LIN {X 0,Y 573.258,Z 350.075,A -85,B 0,C 180,E1 -2304.01,E2 -2304.01} C_VEL
LIN {X 0,Y 573.278,Z 350.069,A -85,B 0,C 180,E1 -2306.518,E2 -2306.518} C_VEL
LIN {X 0,Y 573.237,Z 350.079,A -85,B 0,C 180,E1 -2309.114,E2 -2309.114} C_VEL
LIN {X 0,Y 573.258,Z 350.074,A -85,B 0,C 180,E1 -2311.968,E2 -2311.968} C_VEL
LIN {X 0,Y 573.248,Z 350.071,A -85,B 0,C 180,E1 -2314.59,E2 -2314.59} C_VEL
LIN {X 0,Y 573.251,Z 350.077,A -85,B 0,C 180,E1 -2317.663,E2 -2317.663} C_VEL
LIN {X 0,Y 573.27,Z 350.072,A -85,B 0,C 180,E1 -2320.727,E2 -2320.727} C_VEL
LIN {X 0,Y 573.253,Z 350.076,A -85,B 0,C 180,E1 -2323.622,E2 -2323.622} C_VEL
LIN {X 0,Y 573.232,Z 350.077,A -85,B 0,C 180,E1 -2326.53,E2 -2326.53} C_VEL
LIN {X 0,Y 573.269,Z 350.075,A -85,B 0,C 180,E1 -2329.404,E2 -2329.404} C_VEL
LIN {X 0,Y 573.282,Z 350.069,A -85,B 0,C 180,E1 -2332.25,E2 -2332.25} C_VEL
LIN {X 0,Y 573.307,Z 350.074,A -85,B 0,C 180,E1 -2335.077,E2 -2335.077} C_VEL
LIN {X 0,Y 573.301,Z 350.066,A -85,B 0,C 180,E1 -2337.893,E2 -2337.893} C_VEL
LIN {X 0,Y 573.334,Z 350.07,A -85,B 0,C 180,E1 -2340.703,E2 -2340.703} C_VEL
LIN {X 0,Y 573.237,Z 350.074,A -85,B 0,C 180,E1 -2343.515,E2 -2343.515} C_VEL
LIN {X 0,Y 573.286,Z 350.069,A -85,B 0,C 180,E1 -2345.628,E2 -2345.628} C_VEL
LIN {X 0,Y 573.3,Z 350.072,A -85,B 0,C 180,E1 -2348.459,E2 -2348.459} C_VEL
LIN {X 0,Y 573.29,Z 350.069,A -85,B 0,C 180,E1 -2351.312,E2 -2351.312} C_VEL
LIN {X 0,Y 573.272,Z 350.077,A -85,B 0,C 180,E1 -2354.425,E2 -2354.425} C_VEL
LIN {X 0,Y 573.252,Z 350.074,A -85,B 0,C 180,E1 -2357.112,E2 -2357.112} C_VEL
LIN {X 0,Y 573.249,Z 350.077,A -85,B 0,C 180,E1 -2360.077,E2 -2360.077} C_VEL
LIN {X 0,Y 573.232,Z 350.084,A -85,B 0,C 180,E1 -2362.338,E2 -2362.338} C_VEL
LIN {X 0,Y 573.244,Z 350.076,A -85,B 0,C 180,E1 -2364.406,E2 -2364.406} C_VEL
LIN {X 0,Y 572.619,Z 350.155,A -85,B 0,C 180,E1 -2364.993,E2 -2364.993} C_VEL
LIN {X 0,Y 569.78,Z 350.507,A -85,B 0,C 180,E1 -2365.944,E2 -2365.944} C_VEL
LIN {X 0,Y 567.351,Z 350.81,A -85,B 0,C 180,E1 -2366.71,E2 -2366.71} C_VEL
LIN {X 0,Y 566.299,Z 350.937,A -85,B 0,C 180,E1 -2367.301,E2 -2367.301} C_VEL
LIN {X 0,Y 566.21,Z 350.948,A -85,B 0,C 180,E1 -2367.502,E2 -2367.502} C_VEL
LIN {X 0,Y 566.182,Z 350.957,A -85,B 0,C 180,E1 -2370.593,E2 -2370.593} C_VEL
LIN {X 0,Y 566.224,Z 350.948,A -85,B 0,C 180,E1 -2373.102,E2 -2373.102} C_VEL
LIN {X 0,Y 566.207,Z 350.954,A -85,B 0,C 180,E1 -2375.689,E2 -2375.689} C_VEL
LIN {X 0,Y 566.213,Z 350.953,A -85,B 0,C 180,E1 -2378.56,E2 -2378.56} C_VEL
LIN {X 0,Y 566.21,Z 350.951,A -85,B 0,C 180,E1 -2381.137,E2 -2381.137} C_VEL
LIN {X 0,Y 566.198,Z 350.962,A -85,B 0,C 180,E1 -2384.036,E2 -2384.036} C_VEL
LIN {X 0,Y 566.203,Z 350.952,A -85,B 0,C 180,E1 -2387.083,E2 -2387.083} C_VEL
LIN {X 0,Y 566.227,Z 350.958,A -85,B 0,C 180,E1 -2389.804,E2 -2389.804} C_VEL
LIN {X 0,Y 566.2,Z 350.952,A -85,B 0,C 180,E1 -2392.6,E2 -2392.6} C_VEL
LIN {X 0,Y 566.223,Z 350.951,A -85,B 0,C 180,E1 -2395.184,E2 -2395.184} C_VEL
LIN {X 0,Y 566.234,Z 350.956,A -85,B 0,C 180,E1 -2397.744,E2 -2397.744} C_VEL
LIN {X 0,Y 566.231,Z 350.95,A -85,B 0,C 180,E1 -2400.324,E2 -2400.324} C_VEL
LIN {X 0,Y 566.246,Z 351.051,A -85,B 0,C 180,E1 -2402.588,E2 -2402.588} C_VEL
LIN {X 0,Y 566.363,Z 357.712,A -85,B 0,C 180,E1 -2403.864,E2 -2403.864} C_VEL
LIN {X 0,Y 566.226,Z 372.791,A -85,B 0,C 180,E1 -2406.707,E2 -2406.707} C_VEL
LIN {X 0,Y 566.214,Z 374.601,A -85,B 0,C 180,E1 -2407.046,E2 -2407.046} C_VEL
LIN {X 0,Y 567.183,Z 380.548,A -85,B 0,C 180,E1 -2407.157,E2 -2407.157} C_VEL
LIN {X 0,Y 566.926,Z 481.627,A -85,B 0,C 180,E1 -2408.461,E2 -2408.461} C_VEL
LIN {X 0,Y 566.83,Z 495.188,A -85,B 0,C 180,E1 -2408.793,E2 -2408.793} C_VEL
LIN {X 0,Y 566.692,Z 507.886,A -85,B 0,C 180,E1 -2409.254,E2 -2409.254} C_VEL
LIN {X 0,Y 566.578,Z 520.156,A -85,B 0,C 180,E1 -2409.866,E2 -2409.866} C_VEL
LIN {X 0,Y 566.42,Z 531.079,A -85,B 0,C 180,E1 -2410.561,E2 -2410.561} C_VEL
LIN {X 0,Y 566.291,Z 541.23,A -85,B 0,C 180,E1 -2411.363,E2 -2411.363} C_VEL
LIN {X 0,Y 566.183,Z 550.756,A -85,B 0,C 180,E1 -2412.295,E2 -2412.295} C_VEL
LIN {X 0,Y 566.05,Z 559.938,A -85,B 0,C 180,E1 -2413.408,E2 -2413.408} C_VEL
LIN {X 0,Y 566.009,Z 567.237,A -85,B 0,C 180,E1 -2414.517,E2 -2414.517} C_VEL
LIN {X 0,Y 565.941,Z 572.998,A -85,B 0,C 180,E1 -2415.62,E2 -2415.62} C_VEL
LIN {X 0,Y 565.929,Z 577.491,A -85,B 0,C 180,E1 -2416.718,E2 -2416.718} C_VEL
LIN {X 0,Y 565.895,Z 580.853,A -85,B 0,C 180,E1 -2417.812,E2 -2417.812} C_VEL
LIN {X 0,Y 565.905,Z 583.1,A -85,B 0,C 180,E1 -2418.847,E2 -2418.847} C_VEL
LIN {X 0,Y 565.883,Z 584.554,A -85,B 0,C 180,E1 -2419.987,E2 -2419.987} C_VEL
LIN {X 0,Y 565.853,Z 584.921,A -85,B 0,C 180,E1 -2421.429,E2 -2421.429} C_VEL
LIN {X 0,Y 565.879,Z 584.522,A -85,B 0,C 180,E1 -2422.148,E2 -2422.148} C_VEL
LIN {X 0,Y 565.921,Z 582.681,A -85,B 0,C 180,E1 -2423.466,E2 -2423.466} C_VEL
LIN {X 0,Y 565.917,Z 579.807,A -85,B 0,C 180,E1 -2424.656,E2 -2424.656} C_VEL
LIN {X 0,Y 565.957,Z 576.164,A -85,B 0,C 180,E1 -2425.727,E2 -2425.727} C_VEL
LIN {X 0,Y 565.954,Z 571.425,A -85,B 0,C 180,E1 -2426.797,E2 -2426.797} C_VEL
LIN {X 0,Y 566.008,Z 564.341,A -85,B 0,C 180,E1 -2428.043,E2 -2428.043} C_VEL
LIN {X 0,Y 566.12,Z 556.652,A -85,B 0,C 180,E1 -2429.111,E2 -2429.111} C_VEL
LIN {X 0,Y 566.205,Z 547.068,A -85,B 0,C 180,E1 -2430.178,E2 -2430.178} C_VEL
LIN {X 0,Y 566.344,Z 537.198,A -85,B 0,C 180,E1 -2431.067,E2 -2431.067} C_VEL
LIN {X 0,Y 566.445,Z 526.095,A -85,B 0,C 180,E1 -2431.866,E2 -2431.866} C_VEL
LIN {X 0,Y 566.589,Z 515.253,A -85,B 0,C 180,E1 -2432.488,E2 -2432.488} C_VEL
LIN {X 0,Y 566.707,Z 503.304,A -85,B 0,C 180,E1 -2433.021,E2 -2433.021} C_VEL
LIN {X 0,Y 566.839,Z 490.96,A -85,B 0,C 180,E1 -2433.421,E2 -2433.421} C_VEL
LIN {X 0,Y 566.908,Z 478.202,A -85,B 0,C 180,E1 -2433.687,E2 -2433.687} C_VEL
LIN {X 0,Y 567.109,Z 380.113,A -85,B 0,C 180,E1 -2434.94,E2 -2434.94} C_VEL
LIN {X 0,Y 566.288,Z 374.554,A -85,B 0,C 180,E1 -2435.051,E2 -2435.051} C_VEL
LIN {X 0,Y 566.37,Z 357.828,A -85,B 0,C 180,E1 -2438.204,E2 -2438.204} C_VEL
LIN {X 0,Y 566.223,Z 350.954,A -85,B 0,C 180,E1 -2439.533,E2 -2439.533} C_VEL
LIN {X 0,Y 566.247,Z 350.953,A -85,B 0,C 180,E1 -2442.18,E2 -2442.18} C_VEL
LIN {X 0,Y 566.205,Z 350.951,A -85,B 0,C 180,E1 -2445.109,E2 -2445.109} C_VEL
LIN {X 0,Y 566.205,Z 350.951,A -85,B 0,C 180,E1 -2447.331,E2 -2447.331} C_VEL
LIN {X 0,Y 566.213,Z 350.959,A -85,B 0,C 180,E1 -2450.337,E2 -2450.337} C_VEL
LIN {X 0,Y 566.194,Z 350.952,A -85,B 0,C 180,E1 -2453.403,E2 -2453.403} C_VEL
LIN {X 0,Y 566.217,Z 350.952,A -85,B 0,C 180,E1 -2455.748,E2 -2455.748} C_VEL
LIN {X 0,Y 566.21,Z 350.96,A -85,B 0,C 180,E1 -2458.202,E2 -2458.202} C_VEL
LIN {X 0,Y 566.189,Z 350.956,A -85,B 0,C 180,E1 -2460.591,E2 -2460.591} C_VEL
LIN {X 0,Y 566.23,Z 350.948,A -85,B 0,C 180,E1 -2463.101,E2 -2463.101} C_VEL
LIN {X 0,Y 566.214,Z 350.955,A -85,B 0,C 180,E1 -2465.687,E2 -2465.687} C_VEL
LIN {X 0,Y 566.216,Z 350.951,A -85,B 0,C 180,E1 -2468.558,E2 -2468.558} C_VEL
LIN {X 0,Y 566.202,Z 350.952,A -85,B 0,C 180,E1 -2471.136,E2 -2471.136} C_VEL
LIN {X 0,Y 566.195,Z 350.959,A -85,B 0,C 180,E1 -2474.035,E2 -2474.035} C_VEL
LIN {X 0,Y 566.203,Z 350.952,A -85,B 0,C 180,E1 -2477.081,E2 -2477.081} C_VEL
LIN {X 0,Y 566.223,Z 350.958,A -85,B 0,C 180,E1 -2479.802,E2 -2479.802} C_VEL
LIN {X 0,Y 566.195,Z 350.953,A -85,B 0,C 180,E1 -2482.598,E2 -2482.598} C_VEL
LIN {X 0,Y 566.204,Z 350.954,A -85,B 0,C 180,E1 -2485.181,E2 -2485.181} C_VEL
LIN {X 0,Y 566.231,Z 350.956,A -85,B 0,C 180,E1 -2487.743,E2 -2487.743} C_VEL
LIN {X 0,Y 566.198,Z 350.953,A -85,B 0,C 180,E1 -2490.327,E2 -2490.327} C_VEL
LIN {X 0,Y 566.219,Z 350.95,A -85,B 0,C 180,E1 -2492.661,E2 -2492.661} C_VEL
LIN {X 0,Y 566.228,Z 350.952,A -85,B 0,C 180,E1 -2495.038,E2 -2495.038} C_VEL
LIN {X 0,Y 566.197,Z 350.96,A -85,B 0,C 180,E1 -2497.369,E2 -2497.369} C_VEL
LIN {X 0,Y 566.213,Z 350.956,A -85,B 0,C 180,E1 -2499.663,E2 -2499.663} C_VEL
LIN {X 0,Y 566.198,Z 350.954,A -85,B 0,C 180,E1 -2502.668,E2 -2502.668} C_VEL
LIN {X 0,Y 566.225,Z 350.953,A -85,B 0,C 180,E1 -2505.626,E2 -2505.626} C_VEL
LIN {X 0,Y 566.266,Z 350.946,A -85,B 0,C 180,E1 -2508.654,E2 -2508.654} C_VEL
LIN {X 0,Y 566.242,Z 350.953,A -85,B 0,C 180,E1 -2511.434,E2 -2511.434} C_VEL
LIN {X 0,Y 566.255,Z 350.946,A -85,B 0,C 180,E1 -2514.301,E2 -2514.301} C_VEL
LIN {X 0,Y 566.273,Z 350.943,A -85,B 0,C 180,E1 -2517.866,E2 -2517.866} C_VEL
LIN {X 0,Y 566.302,Z 350.945,A -85,B 0,C 180,E1 -2520.711,E2 -2520.711} C_VEL
LIN {X 0,Y 566.273,Z 350.951,A -85,B 0,C 180,E1 -2522.845,E2 -2522.845} C_VEL
LIN {X 0,Y 566.255,Z 350.946,A -85,B 0,C 180,E1 -2525.698,E2 -2525.698} C_VEL
LIN {X 0,Y 566.241,Z 350.952,A -85,B 0,C 180,E1 -2528.565,E2 -2528.565} C_VEL
LIN {X 0,Y 566.241,Z 350.948,A -85,B 0,C 180,E1 -2531.454,E2 -2531.454} C_VEL
LIN {X 0,Y 566.224,Z 350.955,A -85,B 0,C 180,E1 -2534.507,E2 -2534.507} C_VEL
LIN {X 0,Y 566.197,Z 350.954,A -85,B 0,C 180,E1 -2537.332,E2 -2537.332} C_VEL
LIN {X 0,Y 566.213,Z 350.955,A -85,B 0,C 180,E1 -2540.337,E2 -2540.337} C_VEL
LIN {X 0,Y 566.222,Z 350.95,A -85,B 0,C 180,E1 -2543.402,E2 -2543.402} C_VEL
LIN {X 0,Y 566.217,Z 350.95,A -85,B 0,C 180,E1 -2545.749,E2 -2545.749} C_VEL
LIN {X 0,Y 566.2,Z 350.957,A -85,B 0,C 180,E1 -2548.204,E2 -2548.204} C_VEL
LIN {X 0,Y 566.193,Z 350.954,A -85,B 0,C 180,E1 -2551.079,E2 -2551.079} C_VEL
LIN {X 0,Y 566.222,Z 350.95,A -85,B 0,C 180,E1 -2553.738,E2 -2553.738} C_VEL
LIN {X 0,Y 566.21,Z 350.957,A -85,B 0,C 180,E1 -2556.569,E2 -2556.569} C_VEL
LIN {X 0,Y 566.207,Z 350.952,A -85,B 0,C 180,E1 -2559.686,E2 -2559.686} C_VEL
LIN {X 0,Y 566.209,Z 350.958,A -85,B 0,C 180,E1 -2562.088,E2 -2562.088} C_VEL
LIN {X 0,Y 566.169,Z 350.956,A -85,B 0,C 180,E1 -2565.037,E2 -2565.037} C_VEL
LIN {X 0,Y 566.214,Z 350.959,A -85,B 0,C 180,E1 -2568.137,E2 -2568.137} C_VEL
LIN {X 0,Y 566.22,Z 350.95,A -85,B 0,C 180,E1 -2570.728,E2 -2570.728} C_VEL
LIN {X 0,Y 566.216,Z 350.955,A -85,B 0,C 180,E1 -2573.784,E2 -2573.784} C_VEL
LIN {X 0,Y 566.211,Z 350.955,A -85,B 0,C 180,E1 -2576.266,E2 -2576.266} C_VEL
LIN {X 0,Y 566.202,Z 350.951,A -85,B 0,C 180,E1 -2578.922,E2 -2578.922} C_VEL
LIN {X 0,Y 566.195,Z 350.953,A -85,B 0,C 180,E1 -2581.048,E2 -2581.048} C_VEL
LIN {X 0,Y 566.217,Z 350.954,A -85,B 0,C 180,E1 -2583.46,E2 -2583.46} C_VEL
LIN {X 0,Y 566.236,Z 351.046,A -85,B 0,C 180,E1 -2585.919,E2 -2585.919} C_VEL
LIN {X 0,Y 567.201,Z 357.181,A -85,B 0,C 180,E1 -2586.834,E2 -2586.834} C_VEL
LIN {X 0,Y 566.963,Z 376.072,A -85,B 0,C 180,E1 -2589.502,E2 -2589.502} C_VEL
LIN {X 0,Y 566.667,Z 397.345,A -85,B 0,C 180,E1 -2592.497,E2 -2592.497} C_VEL
LIN {X 0,Y 566.459,Z 419.948,A -85,B 0,C 180,E1 -2595.633,E2 -2595.633} C_VEL
LIN {X 0,Y 566.417,Z 422.524,A -85,B 0,C 180,E1 -2595.987,E2 -2595.987} C_VEL
LIN {X 0,Y 567.226,Z 430.323,A -85,B 0,C 180,E1 -2596.11,E2 -2596.11} C_VEL
LIN {X 0,Y 566.964,Z 530.961,A -85,B 0,C 180,E1 -2597.403,E2 -2597.403} C_VEL
LIN {X 0,Y 566.871,Z 544.228,A -85,B 0,C 180,E1 -2597.72,E2 -2597.72} C_VEL
LIN {X 0,Y 566.74,Z 556.383,A -85,B 0,C 180,E1 -2598.148,E2 -2598.148} C_VEL
LIN {X 0,Y 566.589,Z 568.449,A -85,B 0,C 180,E1 -2598.724,E2 -2598.724} C_VEL
LIN {X 0,Y 566.442,Z 580.203,A -85,B 0,C 180,E1 -2599.455,E2 -2599.455} C_VEL
LIN {X 0,Y 566.321,Z 590.605,A -85,B 0,C 180,E1 -2600.266,E2 -2600.266} C_VEL
LIN {X 0,Y 566.207,Z 599.115,A -85,B 0,C 180,E1 -2601.074,E2 -2601.074} C_VEL
LIN {X 0,Y 566.112,Z 606.962,A -85,B 0,C 180,E1 -2601.972,E2 -2601.972} C_VEL
LIN {X 0,Y 566.003,Z 614.623,A -85,B 0,C 180,E1 -2603.047,E2 -2603.047} C_VEL
LIN {X 0,Y 566.004,Z 621.68,A -85,B 0,C 180,E1 -2604.299,E2 -2604.299} C_VEL
LIN {X 0,Y 565.933,Z 626.373,A -85,B 0,C 180,E1 -2605.37,E2 -2605.37} C_VEL
LIN {X 0,Y 565.927,Z 629.958,A -85,B 0,C 180,E1 -2606.44,E2 -2606.44} C_VEL
LIN {X 0,Y 565.878,Z 631.808,A -85,B 0,C 180,E1 -2607.153,E2 -2607.153} C_VEL
LIN {X 0,Y 565.846,Z 634.185,A -85,B 0,C 180,E1 -2608.577,E2 -2608.577} C_VEL
LIN {X 0,Y 565.839,Z 635,A -85,B 0,C 180,E1 -2610,E2 -2610} C_VEL
LIN {X 0,Y 565.846,Z 634.186,A -85,B 0,C 180,E1 -2611.423,E2 -2611.423} C_VEL
LIN {X 0,Y 565.878,Z 631.81,A -85,B 0,C 180,E1 -2612.847,E2 -2612.847} C_VEL
LIN {X 0,Y 565.926,Z 628.896,A -85,B 0,C 180,E1 -2613.916,E2 -2613.916} C_VEL
LIN {X 0,Y 565.878,Z 624.949,A -85,B 0,C 180,E1 -2614.987,E2 -2614.987} C_VEL
LIN {X 0,Y 566.002,Z 619.868,A -85,B 0,C 180,E1 -2616.058,E2 -2616.058} C_VEL
LIN {X 0,Y 566.04,Z 613.469,A -85,B 0,C 180,E1 -2617.132,E2 -2617.132} C_VEL
LIN {X 0,Y 566.133,Z 605.479,A -85,B 0,C 180,E1 -2618.207,E2 -2618.207} C_VEL
LIN {X 0,Y 566.228,Z 597.337,A -85,B 0,C 180,E1 -2619.105,E2 -2619.105} C_VEL
LIN {X 0,Y 566.343,Z 587.403,A -85,B 0,C 180,E1 -2620.005,E2 -2620.005} C_VEL
LIN {X 0,Y 566.529,Z 576.294,A -85,B 0,C 180,E1 -2620.807,E2 -2620.807} C_VEL
LIN {X 0,Y 566.612,Z 565.181,A -85,B 0,C 180,E1 -2621.446,E2 -2621.446} C_VEL
LIN {X 0,Y 566.736,Z 552.989,A -85,B 0,C 180,E1 -2621.988,E2 -2621.988} C_VEL
LIN {X 0,Y 566.91,Z 540.187,A -85,B 0,C 180,E1 -2622.393,E2 -2622.393} C_VEL
LIN {X 0,Y 566.997,Z 528.125,A -85,B 0,C 180,E1 -2622.641,E2 -2622.641} C_VEL
LIN {X 0,Y 567.065,Z 426.951,A -85,B 0,C 180,E1 -2623.937,E2 -2623.937} C_VEL
LIN {X 0,Y 566.435,Z 422.441,A -85,B 0,C 180,E1 -2624.024,E2 -2624.024} C_VEL
LIN {X 0,Y 566.648,Z 399.148,A -85,B 0,C 180,E1 -2627.251,E2 -2627.251} C_VEL
LIN {X 0,Y 566.926,Z 378.732,A -85,B 0,C 180,E1 -2630.121,E2 -2630.121} C_VEL
LIN {X 0,Y 567.199,Z 357.121,A -85,B 0,C 180,E1 -2633.166,E2 -2633.166} C_VEL
LIN {X 0,Y 566.236,Z 350.957,A -85,B 0,C 180,E1 -2634.105,E2 -2634.105} C_VEL
LIN {X 0,Y 566.209,Z 350.954,A -85,B 0,C 180,E1 -2636.659,E2 -2636.659} C_VEL
LIN {X 0,Y 566.195,Z 350.953,A -85,B 0,C 180,E1 -2638.952,E2 -2638.952} C_VEL
LIN {X 0,Y 566.202,Z 350.952,A -85,B 0,C 180,E1 -2641.42,E2 -2641.42} C_VEL
LIN {X 0,Y 566.211,Z 350.959,A -85,B 0,C 180,E1 -2643.955,E2 -2643.955} C_VEL
LIN {X 0,Y 566.215,Z 350.951,A -85,B 0,C 180,E1 -2646.568,E2 -2646.568} C_VEL
LIN {X 0,Y 566.21,Z 350.957,A -85,B 0,C 180,E1 -2649.685,E2 -2649.685} C_VEL
LIN {X 0,Y 566.209,Z 350.955,A -85,B 0,C 180,E1 -2652.087,E2 -2652.087} C_VEL
LIN {X 0,Y 566.169,Z 350.955,A -85,B 0,C 180,E1 -2655.035,E2 -2655.035} C_VEL
LIN {X 0,Y 566.209,Z 350.956,A -85,B 0,C 180,E1 -2657.912,E2 -2657.912} C_VEL
LIN {X 0,Y 566.216,Z 350.949,A -85,B 0,C 180,E1 -2660.726,E2 -2660.726} C_VEL
LIN {X 0,Y 566.211,Z 350.956,A -85,B 0,C 180,E1 -2663.783,E2 -2663.783} C_VEL
LIN {X 0,Y 566.222,Z 350.949,A -85,B 0,C 180,E1 -2666.262,E2 -2666.262} C_VEL
LIN {X 0,Y 566.196,Z 350.954,A -85,B 0,C 180,E1 -2668.921,E2 -2668.921} C_VEL
LIN {X 0,Y 566.191,Z 350.956,A -85,B 0,C 180,E1 -2671.047,E2 -2671.047} C_VEL
LIN {X 0,Y 566.239,Z 350.953,A -85,B 0,C 180,E1 -2673.46,E2 -2673.46} C_VEL
LIN {X 0,Y 566.197,Z 350.953,A -85,B 0,C 180,E1 -2675.819,E2 -2675.819} C_VEL
LIN {X 0,Y 566.209,Z 350.954,A -85,B 0,C 180,E1 -2678.902,E2 -2678.902} C_VEL
LIN {X 0,Y 566.206,Z 350.959,A -85,B 0,C 180,E1 -2681.172,E2 -2681.172} C_VEL
LIN {X 0,Y 566.215,Z 350.955,A -85,B 0,C 180,E1 -2683.412,E2 -2683.412} C_VEL
LIN {X 0,Y 566.194,Z 350.952,A -85,B 0,C 180,E1 -2686.359,E2 -2686.359} C_VEL
LIN {X 0,Y 566.265,Z 350.946,A -85,B 0,C 180,E1 -2688.654,E2 -2688.654} C_VEL
LIN {X 0,Y 566.242,Z 350.95,A -85,B 0,C 180,E1 -2691.435,E2 -2691.435} C_VEL
LIN {X 0,Y 566.255,Z 350.944,A -85,B 0,C 180,E1 -2694.302,E2 -2694.302} C_VEL
LIN {X 0,Y 566.272,Z 350.942,A -85,B 0,C 180,E1 -2697.866,E2 -2697.866} C_VEL
LIN {X 0,Y 566.303,Z 350.946,A -85,B 0,C 180,E1 -2700.711,E2 -2700.711} C_VEL
LIN {X 0,Y 566.274,Z 350.95,A -85,B 0,C 180,E1 -2702.846,E2 -2702.846} C_VEL
LIN {X 0,Y 566.254,Z 350.945,A -85,B 0,C 180,E1 -2705.699,E2 -2705.699} C_VEL
LIN {X 0,Y 566.241,Z 350.953,A -85,B 0,C 180,E1 -2708.566,E2 -2708.566} C_VEL
LIN {X 0,Y 566.242,Z 350.946,A -85,B 0,C 180,E1 -2711.455,E2 -2711.455} C_VEL
LIN {X 0,Y 566.225,Z 350.957,A -85,B 0,C 180,E1 -2714.507,E2 -2714.507} C_VEL
LIN {X 0,Y 566.196,Z 350.951,A -85,B 0,C 180,E1 -2717.332,E2 -2717.332} C_VEL
LIN {X 0,Y 566.212,Z 350.958,A -85,B 0,C 180,E1 -2720.338,E2 -2720.338} C_VEL
LIN {X 0,Y 566.182,Z 350.953,A -85,B 0,C 180,E1 -2723.405,E2 -2723.405} C_VEL
LIN {X 0,Y 566.218,Z 350.949,A -85,B 0,C 180,E1 -2725.749,E2 -2725.749} C_VEL
LIN {X 0,Y 566.21,Z 350.948,A -85,B 0,C 180,E1 -2727.502,E2 -2727.502} C_VEL
LIN {X 0,Y 565.531,Z 351.041,A -85,B 0,C 180,E1 -2728.095,E2 -2728.095} C_VEL
LIN {X 0,Y 562.66,Z 351.399,A -85,B 0,C 180,E1 -2729.059,E2 -2729.059} C_VEL
LIN {X 0,Y 560.245,Z 351.7,A -85,B 0,C 180,E1 -2729.834,E2 -2729.834} C_VEL
LIN {X 0,Y 559.218,Z 351.827,A -85,B 0,C 180,E1 -2730.433,E2 -2730.433} C_VEL
LIN {X 0,Y 559.139,Z 351.833,A -85,B 0,C 180,E1 -2730.636,E2 -2730.636} C_VEL
LIN {X 0,Y 559.16,Z 351.83,A -85,B 0,C 180,E1 -2733.576,E2 -2733.576} C_VEL
LIN {X 0,Y 559.165,Z 351.832,A -85,B 0,C 180,E1 -2736.45,E2 -2736.45} C_VEL
LIN {X 0,Y 559.175,Z 351.827,A -85,B 0,C 180,E1 -2738.935,E2 -2738.935} C_VEL
LIN {X 0,Y 559.19,Z 351.831,A -85,B 0,C 180,E1 -2741.768,E2 -2741.768} C_VEL
LIN {X 0,Y 559.138,Z 351.833,A -85,B 0,C 180,E1 -2744.74,E2 -2744.74} C_VEL
LIN {X 0,Y 559.162,Z 351.83,A -85,B 0,C 180,E1 -2747.258,E2 -2747.258} C_VEL
LIN {X 0,Y 559.187,Z 351.831,A -85,B 0,C 180,E1 -2750.136,E2 -2750.136} C_VEL
LIN {X 0,Y 559.148,Z 351.831,A -85,B 0,C 180,E1 -2752.893,E2 -2752.893} C_VEL
LIN {X 0,Y 559.159,Z 351.836,A -85,B 0,C 180,E1 -2755.557,E2 -2755.557} C_VEL
LIN {X 0,Y 559.169,Z 351.832,A -85,B 0,C 180,E1 -2758.138,E2 -2758.138} C_VEL
LIN {X 0,Y 559.16,Z 351.83,A -85,B 0,C 180,E1 -2760.648,E2 -2760.648} C_VEL
LIN {X 0,Y 559.233,Z 351.926,A -85,B 0,C 180,E1 -2762.494,E2 -2762.494} C_VEL
LIN {X 0,Y 559.331,Z 359.115,A -85,B 0,C 180,E1 -2763.911,E2 -2763.911} C_VEL
LIN {X 0,Y 559.188,Z 374.319,A -85,B 0,C 180,E1 -2766.813,E2 -2766.813} C_VEL
LIN {X 0,Y 559.178,Z 374.608,A -85,B 0,C 180,E1 -2766.868,E2 -2766.868} C_VEL
LIN {X 0,Y 560.329,Z 382.548,A -85,B 0,C 180,E1 -2767.01,E2 -2767.01} C_VEL
LIN {X 0,Y 560.014,Z 480.749,A -85,B 0,C 180,E1 -2768.285,E2 -2768.285} C_VEL
LIN {X 0,Y 559.889,Z 494.348,A -85,B 0,C 180,E1 -2768.613,E2 -2768.613} C_VEL
LIN {X 0,Y 559.752,Z 507.31,A -85,B 0,C 180,E1 -2769.081,E2 -2769.081} C_VEL
LIN {X 0,Y 559.609,Z 519.727,A -85,B 0,C 180,E1 -2769.701,E2 -2769.701} C_VEL
LIN {X 0,Y 559.436,Z 531.035,A -85,B 0,C 180,E1 -2770.426,E2 -2770.426} C_VEL
LIN {X 0,Y 559.272,Z 542.001,A -85,B 0,C 180,E1 -2771.311,E2 -2771.311} C_VEL
LIN {X 0,Y 559.136,Z 551.377,A -85,B 0,C 180,E1 -2772.254,E2 -2772.254} C_VEL
LIN {X 0,Y 559.015,Z 559.056,A -85,B 0,C 180,E1 -2773.193,E2 -2773.193} C_VEL
LIN {X 0,Y 558.904,Z 566.544,A -85,B 0,C 180,E1 -2774.315,E2 -2774.315} C_VEL
LIN {X 0,Y 558.851,Z 572.974,A -85,B 0,C 180,E1 -2775.545,E2 -2775.545} C_VEL
LIN {X 0,Y 558.808,Z 578.359,A -85,B 0,C 180,E1 -2776.916,E2 -2776.916} C_VEL
LIN {X 0,Y 558.806,Z 580.566,A -85,B 0,C 180,E1 -2777.655,E2 -2777.655} C_VEL
LIN {X 0,Y 558.802,Z 583.093,A -85,B 0,C 180,E1 -2778.816,E2 -2778.816} C_VEL
LIN {X 0,Y 558.779,Z 584.462,A -85,B 0,C 180,E1 -2779.859,E2 -2779.859} C_VEL
LIN {X 0,Y 558.741,Z 584.906,A -85,B 0,C 180,E1 -2780.589,E2 -2780.589} C_VEL
LIN {X 0,Y 558.797,Z 584.599,A -85,B 0,C 180,E1 -2782.048,E2 -2782.048} C_VEL
LIN {X 0,Y 558.797,Z 583.858,A -85,B 0,C 180,E1 -2782.775,E2 -2782.775} C_VEL
LIN {X 0,Y 558.828,Z 582.673,A -85,B 0,C 180,E1 -2783.501,E2 -2783.501} C_VEL
LIN {X 0,Y 558.839,Z 580.14,A -85,B 0,C 180,E1 -2784.588,E2 -2784.588} C_VEL
LIN {X 0,Y 558.861,Z 576.612,A -85,B 0,C 180,E1 -2785.673,E2 -2785.673} C_VEL
LIN {X 0,Y 558.874,Z 571.993,A -85,B 0,C 180,E1 -2786.756,E2 -2786.756} C_VEL
LIN {X 0,Y 558.919,Z 565.045,A -85,B 0,C 180,E1 -2788.018,E2 -2788.018} C_VEL
LIN {X 0,Y 559.063,Z 557.541,A -85,B 0,C 180,E1 -2789.1,E2 -2789.1} C_VEL
LIN {X 0,Y 559.122,Z 549.916,A -85,B 0,C 180,E1 -2790,E2 -2790} C_VEL
LIN {X 0,Y 559.309,Z 539.588,A -85,B 0,C 180,E1 -2790.99,E2 -2790.99} C_VEL
LIN {X 0,Y 559.416,Z 529.127,A -85,B 0,C 180,E1 -2791.8,E2 -2791.8} C_VEL
LIN {X 0,Y 559.586,Z 517.436,A -85,B 0,C 180,E1 -2792.519,E2 -2792.519} C_VEL
LIN {X 0,Y 559.733,Z 504.991,A -85,B 0,C 180,E1 -2793.104,E2 -2793.104} C_VEL
LIN {X 0,Y 559.898,Z 491.824,A -85,B 0,C 180,E1 -2793.553,E2 -2793.553} C_VEL
LIN {X 0,Y 559.987,Z 479.715,A -85,B 0,C 180,E1 -2793.823,E2 -2793.823} C_VEL
LIN {X 0,Y 560.192,Z 380.855,A -85,B 0,C 180,E1 -2795.106,E2 -2795.106} C_VEL
LIN {X 0,Y 559.262,Z 374.57,A -85,B 0,C 180,E1 -2795.227,E2 -2795.227} C_VEL
LIN {X 0,Y 559.361,Z 358.442,A -85,B 0,C 180,E1 -2798.308,E2 -2798.308} C_VEL
LIN {X 0,Y 559.182,Z 351.872,A -85,B 0,C 180,E1 -2799.609,E2 -2799.609} C_VEL
LIN {X 0,Y 559.202,Z 351.833,A -85,B 0,C 180,E1 -2802.336,E2 -2802.336} C_VEL
LIN {X 0,Y 559.154,Z 351.829,A -85,B 0,C 180,E1 -2805.304,E2 -2805.304} C_VEL
LIN {X 0,Y 559.164,Z 351.828,A -85,B 0,C 180,E1 -2807.556,E2 -2807.556} C_VEL
LIN {X 0,Y 559.171,Z 351.83,A -85,B 0,C 180,E1 -2809.837,E2 -2809.837} C_VEL
LIN {X 0,Y 559.146,Z 351.838,A -85,B 0,C 180,E1 -2812.152,E2 -2812.152} C_VEL
LIN {X 0,Y 559.183,Z 351.826,A -85,B 0,C 180,E1 -2815.186,E2 -2815.186} C_VEL
LIN {X 0,Y 559.195,Z 351.827,A -85,B 0,C 180,E1 -2817.711,E2 -2817.711} C_VEL
LIN {X 0,Y 559.168,Z 351.836,A -85,B 0,C 180,E1 -2820.181,E2 -2820.181} C_VEL
LIN {X 0,Y 559.176,Z 351.828,A -85,B 0,C 180,E1 -2822.713,E2 -2822.713} C_VEL
LIN {X 0,Y 559.159,Z 351.83,A -85,B 0,C 180,E1 -2825.321,E2 -2825.321} C_VEL
LIN {X 0,Y 559.135,Z 351.841,A -85,B 0,C 180,E1 -2828.016,E2 -2828.016} C_VEL
LIN {X 0,Y 559.172,Z 351.827,A -85,B 0,C 180,E1 -2830.81,E2 -2830.81} C_VEL
LIN {X 0,Y 559.139,Z 351.839,A -85,B 0,C 180,E1 -2833.733,E2 -2833.733} C_VEL
LIN {X 0,Y 559.166,Z 351.828,A -85,B 0,C 180,E1 -2836.8,E2 -2836.8} C_VEL
LIN {X 0,Y 559.173,Z 351.829,A -85,B 0,C 180,E1 -2839.189,E2 -2839.189} C_VEL
LIN {X 0,Y 559.131,Z 351.838,A -85,B 0,C 180,E1 -2841.982,E2 -2841.982} C_VEL
LIN {X 0,Y 559.142,Z 351.831,A -85,B 0,C 180,E1 -2844.784,E2 -2844.784} C_VEL
LIN {X 0,Y 559.17,Z 351.834,A -85,B 0,C 180,E1 -2847.36,E2 -2847.36} C_VEL
LIN {X 0,Y 559.143,Z 351.833,A -85,B 0,C 180,E1 -2850.141,E2 -2850.141} C_VEL
LIN {X 0,Y 559.173,Z 351.831,A -85,B 0,C 180,E1 -2853.097,E2 -2853.097} C_VEL
LIN {X 0,Y 559.154,Z 351.838,A -85,B 0,C 180,E1 -2855.494,E2 -2855.494} C_VEL
LIN {X 0,Y 559.157,Z 351.83,A -85,B 0,C 180,E1 -2858.447,E2 -2858.447} C_VEL
LIN {X 0,Y 559.165,Z 351.832,A -85,B 0,C 180,E1 -2860.926,E2 -2860.926} C_VEL
LIN {X 0,Y 559.166,Z 351.83,A -85,B 0,C 180,E1 -2863.948,E2 -2863.948} C_VEL
LIN {X 0,Y 559.167,Z 351.828,A -85,B 0,C 180,E1 -2866.184,E2 -2866.184} C_VEL
LIN {X 0,Y 559.203,Z 351.831,A -85,B 0,C 180,E1 -2869.133,E2 -2869.133} C_VEL
LIN {X 0,Y 559.205,Z 351.824,A -85,B 0,C 180,E1 -2872.053,E2 -2872.053} C_VEL
LIN {X 0,Y 559.253,Z 351.825,A -85,B 0,C 180,E1 -2874.953,E2 -2874.953} C_VEL
LIN {X 0,Y 559.244,Z 351.819,A -85,B 0,C 180,E1 -2877.839,E2 -2877.839} C_VEL
LIN {X 0,Y 559.272,Z 351.821,A -85,B 0,C 180,E1 -2880.72,E2 -2880.72} C_VEL
LIN {X 0,Y 559.239,Z 351.827,A -85,B 0,C 180,E1 -2882.881,E2 -2882.881} C_VEL
LIN {X 0,Y 559.224,Z 351.822,A -85,B 0,C 180,E1 -2885.77,E2 -2885.77} C_VEL
LIN {X 0,Y 559.196,Z 351.832,A -85,B 0,C 180,E1 -2888.674,E2 -2888.674} C_VEL
LIN {X 0,Y 559.2,Z 351.825,A -85,B 0,C 180,E1 -2891.6,E2 -2891.6} C_VEL
LIN {X 0,Y 559.189,Z 351.833,A -85,B 0,C 180,E1 -2894.596,E2 -2894.596} C_VEL
LIN {X 0,Y 559.156,Z 351.83,A -85,B 0,C 180,E1 -2897.557,E2 -2897.557} C_VEL
LIN {X 0,Y 559.167,Z 351.829,A -85,B 0,C 180,E1 -2899.838,E2 -2899.838} C_VEL
LIN {X 0,Y 559.148,Z 351.834,A -85,B 0,C 180,E1 -2902.152,E2 -2902.152} C_VEL
LIN {X 0,Y 559.153,Z 351.839,A -85,B 0,C 180,E1 -2904.505,E2 -2904.505} C_VEL
LIN {X 0,Y 559.172,Z 351.831,A -85,B 0,C 180,E1 -2906.902,E2 -2906.902} C_VEL
LIN {X 0,Y 559.142,Z 351.833,A -85,B 0,C 180,E1 -2909.858,E2 -2909.858} C_VEL
LIN {X 0,Y 559.169,Z 351.833,A -85,B 0,C 180,E1 -2912.714,E2 -2912.714} C_VEL
LIN {X 0,Y 559.15,Z 351.83,A -85,B 0,C 180,E1 -2915.322,E2 -2915.322} C_VEL
LIN {X 0,Y 559.129,Z 351.838,A -85,B 0,C 180,E1 -2918.018,E2 -2918.018} C_VEL
LIN {X 0,Y 559.171,Z 351.829,A -85,B 0,C 180,E1 -2920.811,E2 -2920.811} C_VEL
LIN {X 0,Y 559.158,Z 351.832,A -85,B 0,C 180,E1 -2923.732,E2 -2923.732} C_VEL
LIN {X 0,Y 559.142,Z 351.832,A -85,B 0,C 180,E1 -2926.804,E2 -2926.804} C_VEL
LIN {X 0,Y 559.173,Z 351.827,A -85,B 0,C 180,E1 -2929.19,E2 -2929.19} C_VEL
LIN {X 0,Y 559.133,Z 351.841,A -85,B 0,C 180,E1 -2931.983,E2 -2931.983} C_VEL
LIN {X 0,Y 559.159,Z 351.829,A -85,B 0,C 180,E1 -2934.784,E2 -2934.784} C_VEL
LIN {X 0,Y 559.173,Z 351.828,A -85,B 0,C 180,E1 -2937.362,E2 -2937.362} C_VEL
LIN {X 0,Y 559.189,Z 351.832,A -85,B 0,C 180,E1 -2940.136,E2 -2940.136} C_VEL
LIN {X 0,Y 559.172,Z 351.829,A -85,B 0,C 180,E1 -2943.173,E2 -2943.173} C_VEL
LIN {X 0,Y 559.2,Z 351.975,A -85,B 0,C 180,E1 -2945.769,E2 -2945.769} C_VEL
LIN {X 0,Y 560.282,Z 358.284,A -85,B 0,C 180,E1 -2946.727,E2 -2946.727} C_VEL
LIN {X 0,Y 560.017,Z 377.22,A -85,B 0,C 180,E1 -2949.428,E2 -2949.428} C_VEL
LIN {X 0,Y 559.713,Z 397.345,A -85,B 0,C 180,E1 -2952.273,E2 -2952.273} C_VEL
LIN {X 0,Y 559.463,Z 418.899,A -85,B 0,C 180,E1 -2955.303,E2 -2955.303} C_VEL
LIN {X 0,Y 559.419,Z 422.524,A -85,B 0,C 180,E1 -2955.808,E2 -2955.808} C_VEL
LIN {X 0,Y 560.336,Z 430.323,A -85,B 0,C 180,E1 -2955.936,E2 -2955.936} C_VEL
LIN {X 0,Y 560.058,Z 530.961,A -85,B 0,C 180,E1 -2957.246,E2 -2957.246} C_VEL
LIN {X 0,Y 559.927,Z 544.227,A -85,B 0,C 180,E1 -2957.565,E2 -2957.565} C_VEL
LIN {X 0,Y 559.786,Z 556.384,A -85,B 0,C 180,E1 -2957.999,E2 -2957.999} C_VEL
LIN {X 0,Y 559.615,Z 568.322,A -85,B 0,C 180,E1 -2958.574,E2 -2958.574} C_VEL
LIN {X 0,Y 559.461,Z 580.201,A -85,B 0,C 180,E1 -2959.322,E2 -2959.322} C_VEL
LIN {X 0,Y 559.301,Z 590.606,A -85,B 0,C 180,E1 -2960.142,E2 -2960.142} C_VEL
LIN {X 0,Y 559.161,Z 599.115,A -85,B 0,C 180,E1 -2960.961,E2 -2960.961} C_VEL
LIN {X 0,Y 559.05,Z 606.962,A -85,B 0,C 180,E1 -2961.87,E2 -2961.87} C_VEL
LIN {X 0,Y 558.943,Z 614.623,A -85,B 0,C 180,E1 -2962.959,E2 -2962.959} C_VEL
LIN {X 0,Y 558.935,Z 621.68,A -85,B 0,C 180,E1 -2964.227,E2 -2964.227} C_VEL
LIN {X 0,Y 558.827,Z 626.373,A -85,B 0,C 180,E1 -2965.311,E2 -2965.311} C_VEL
LIN {X 0,Y 558.836,Z 629.958,A -85,B 0,C 180,E1 -2966.395,E2 -2966.395} C_VEL
LIN {X 0,Y 558.799,Z 631.808,A -85,B 0,C 180,E1 -2967.116,E2 -2967.116} C_VEL
LIN {X 0,Y 558.745,Z 634.184,A -85,B 0,C 180,E1 -2968.559,E2 -2968.559} C_VEL
LIN {X 0,Y 558.74,Z 635,A -85,B 0,C 180,E1 -2970,E2 -2970} C_VEL
LIN {X 0,Y 558.745,Z 634.185,A -85,B 0,C 180,E1 -2971.441,E2 -2971.441} C_VEL
LIN {X 0,Y 558.799,Z 631.81,A -85,B 0,C 180,E1 -2972.884,E2 -2972.884} C_VEL
LIN {X 0,Y 558.843,Z 628.896,A -85,B 0,C 180,E1 -2973.966,E2 -2973.966} C_VEL
LIN {X 0,Y 558.799,Z 624.949,A -85,B 0,C 180,E1 -2975.051,E2 -2975.051} C_VEL
LIN {X 0,Y 558.921,Z 619.868,A -85,B 0,C 180,E1 -2976.135,E2 -2976.135} C_VEL
LIN {X 0,Y 558.977,Z 613.469,A -85,B 0,C 180,E1 -2977.223,E2 -2977.223} C_VEL
LIN {X 0,Y 559.098,Z 605.479,A -85,B 0,C 180,E1 -2978.311,E2 -2978.311} C_VEL
LIN {X 0,Y 559.184,Z 597.337,A -85,B 0,C 180,E1 -2979.221,E2 -2979.221} C_VEL
LIN {X 0,Y 559.356,Z 587.402,A -85,B 0,C 180,E1 -2980.131,E2 -2980.131} C_VEL
LIN {X 0,Y 559.543,Z 576.403,A -85,B 0,C 180,E1 -2980.937,E2 -2980.937} C_VEL
LIN {X 0,Y 559.671,Z 564.465,A -85,B 0,C 180,E1 -2981.627,E2 -2981.627} C_VEL
LIN {X 0,Y 559.817,Z 551.776,A -85,B 0,C 180,E1 -2982.184,E2 -2982.184} C_VEL
LIN {X 0,Y 559.973,Z 538.358,A -85,B 0,C 180,E1 -2982.595,E2 -2982.595} C_VEL
LIN {X 0,Y 560.106,Z 525.105,A -85,B 0,C 180,E1 -2982.845,E2 -2982.845} C_VEL
LIN {X 0,Y 560.246,Z 428.089,A -85,B 0,C 180,E1 -2984.095,E2 -2984.095} C_VEL
LIN {X 0,Y 559.427,Z 422.441,A -85,B 0,C 180,E1 -2984.203,E2 -2984.203} C_VEL
LIN {X 0,Y 559.682,Z 399.799,A -85,B 0,C 180,E1 -2987.38,E2 -2987.38} C_VEL
LIN {X 0,Y 559.962,Z 379.892,A -85,B 0,C 180,E1 -2990.19,E2 -2990.19} C_VEL
LIN {X 0,Y 560.278,Z 358.197,A -85,B 0,C 180,E1 -2993.273,E2 -2993.273} C_VEL
LIN {X 0,Y 559.191,Z 351.834,A -85,B 0,C 180,E1 -2994.256,E2 -2994.256} C_VEL
LIN {X 0,Y 559.171,Z 351.829,A -85,B 0,C 180,E1 -2996.902,E2 -2996.902} C_VEL
LIN {X 0,Y 559.189,Z 351.832,A -85,B 0,C 180,E1 -2999.864,E2 -2999.864} C_VEL
LIN {X 0,Y 559.174,Z 351.828,A -85,B 0,C 180,E1 -3002.713,E2 -3002.713} C_VEL
LIN {X 0,Y 559.157,Z 351.831,A -85,B 0,C 180,E1 -3005.321,E2 -3005.321} C_VEL
LIN {X 0,Y 559.133,Z 351.84,A -85,B 0,C 180,E1 -3008.017,E2 -3008.017} C_VEL
LIN {X 0,Y 559.173,Z 351.826,A -85,B 0,C 180,E1 -3010.81,E2 -3010.81} C_VEL
LIN {X 0,Y 559.155,Z 351.837,A -85,B 0,C 180,E1 -3013.731,E2 -3013.731} C_VEL
LIN {X 0,Y 559.163,Z 351.827,A -85,B 0,C 180,E1 -3016.8,E2 -3016.8} C_VEL
LIN {X 0,Y 559.171,Z 351.829,A -85,B 0,C 180,E1 -3019.189,E2 -3019.189} C_VEL
LIN {X 0,Y 559.13,Z 351.836,A -85,B 0,C 180,E1 -3021.982,E2 -3021.982} C_VEL
LIN {X 0,Y 559.151,Z 351.829,A -85,B 0,C 180,E1 -3024.678,E2 -3024.678} C_VEL
LIN {X 0,Y 559.168,Z 351.834,A -85,B 0,C 180,E1 -3027.36,E2 -3027.36} C_VEL
LIN {X 0,Y 559.182,Z 351.826,A -85,B 0,C 180,E1 -3030.134,E2 -3030.134} C_VEL
LIN {X 0,Y 559.175,Z 351.832,A -85,B 0,C 180,E1 -3033.169,E2 -3033.169} C_VEL
LIN {X 0,Y 559.153,Z 351.835,A -85,B 0,C 180,E1 -3035.495,E2 -3035.495} C_VEL
LIN {X 0,Y 559.156,Z 351.829,A -85,B 0,C 180,E1 -3038.447,E2 -3038.447} C_VEL
LIN {X 0,Y 559.164,Z 351.832,A -85,B 0,C 180,E1 -3040.926,E2 -3040.926} C_VEL
LIN {X 0,Y 559.165,Z 351.828,A -85,B 0,C 180,E1 -3043.948,E2 -3043.948} C_VEL
LIN {X 0,Y 559.167,Z 351.827,A -85,B 0,C 180,E1 -3046.184,E2 -3046.184} C_VEL
LIN {X 0,Y 559.224,Z 351.828,A -85,B 0,C 180,E1 -3049.134,E2 -3049.134} C_VEL
LIN {X 0,Y 559.205,Z 351.823,A -85,B 0,C 180,E1 -3052.054,E2 -3052.054} C_VEL
LIN {X 0,Y 559.253,Z 351.825,A -85,B 0,C 180,E1 -3054.953,E2 -3054.953} C_VEL
LIN {X 0,Y 559.244,Z 351.817,A -85,B 0,C 180,E1 -3057.84,E2 -3057.84} C_VEL
LIN {X 0,Y 559.272,Z 351.822,A -85,B 0,C 180,E1 -3060.72,E2 -3060.72} C_VEL
LIN {X 0,Y 559.239,Z 351.826,A -85,B 0,C 180,E1 -3062.882,E2 -3062.882} C_VEL
LIN {X 0,Y 559.223,Z 351.821,A -85,B 0,C 180,E1 -3065.77,E2 -3065.77} C_VEL
LIN {X 0,Y 559.196,Z 351.832,A -85,B 0,C 180,E1 -3068.674,E2 -3068.674} C_VEL
LIN {X 0,Y 559.2,Z 351.823,A -85,B 0,C 180,E1 -3071.601,E2 -3071.601} C_VEL
LIN {X 0,Y 559.19,Z 351.834,A -85,B 0,C 180,E1 -3074.596,E2 -3074.596} C_VEL
LIN {X 0,Y 559.156,Z 351.828,A -85,B 0,C 180,E1 -3077.557,E2 -3077.557} C_VEL
LIN {X 0,Y 559.167,Z 351.829,A -85,B 0,C 180,E1 -3079.838,E2 -3079.838} C_VEL
LIN {X 0,Y 559.136,Z 351.836,A -85,B 0,C 180,E1 -3082.153,E2 -3082.153} C_VEL
LIN {X 0,Y 559.172,Z 351.825,A -85,B 0,C 180,E1 -3085.188,E2 -3085.188} C_VEL
LIN {X 0,Y 559.188,Z 351.824,A -85,B 0,C 180,E1 -3087.712,E2 -3087.712} C_VEL
LIN {X 0,Y 559.139,Z 351.833,A -85,B 0,C 180,E1 -3090.636,E2 -3090.636} C_VEL
LIN {X 0,Y 558.481,Z 351.915,A -85,B 0,C 180,E1 -3091.237,E2 -3091.237} C_VEL
LIN {X 0,Y 555.619,Z 352.279,A -85,B 0,C 180,E1 -3092.213,E2 -3092.213} C_VEL
LIN {X 0,Y 553.205,Z 352.574,A -85,B 0,C 180,E1 -3092.999,E2 -3092.999} C_VEL
LIN {X 0,Y 552.184,Z 352.7,A -85,B 0,C 180,E1 -3093.606,E2 -3093.606} C_VEL
LIN {X 0,Y 552.11,Z 352.711,A -85,B 0,C 180,E1 -3093.811,E2 -3093.811} C_VEL
LIN {X 0,Y 552.108,Z 352.708,A -85,B 0,C 180,E1 -3096.747,E2 -3096.747} C_VEL
LIN {X 0,Y 552.131,Z 352.706,A -85,B 0,C 180,E1 -3099.528,E2 -3099.528} C_VEL
LIN {X 0,Y 552.128,Z 352.708,A -85,B 0,C 180,E1 -3102.426,E2 -3102.426} C_VEL
LIN {X 0,Y 552.098,Z 352.714,A -85,B 0,C 180,E1 -3105.564,E2 -3105.564} C_VEL
LIN {X 0,Y 552.14,Z 352.705,A -85,B 0,C 180,E1 -3108.677,E2 -3108.677} C_VEL
LIN {X 0,Y 552.121,Z 352.71,A -85,B 0,C 180,E1 -3111.412,E2 -3111.412} C_VEL
LIN {X 0,Y 552.115,Z 352.711,A -85,B 0,C 180,E1 -3114.159,E2 -3114.159} C_VEL
LIN {X 0,Y 552.125,Z 352.706,A -85,B 0,C 180,E1 -3116.816,E2 -3116.816} C_VEL
LIN {X 0,Y 552.144,Z 352.71,A -85,B 0,C 180,E1 -3119.946,E2 -3119.946} C_VEL
LIN {X 0,Y 552.179,Z 352.77,A -85,B 0,C 180,E1 -3122.37,E2 -3122.37} C_VEL
LIN {X 0,Y 552.403,Z 358.674,A -85,B 0,C 180,E1 -3123.559,E2 -3123.559} C_VEL
LIN {X 0,Y 552.158,Z 374.642,A -85,B 0,C 180,E1 -3126.69,E2 -3126.69} C_VEL
LIN {X 0,Y 553.447,Z 383.433,A -85,B 0,C 180,E1 -3126.843,E2 -3126.843} C_VEL
LIN {X 0,Y 553.09,Z 481.472,A -85,B 0,C 180,E1 -3128.138,E2 -3128.138} C_VEL
LIN {X 0,Y 552.957,Z 494.852,A -85,B 0,C 180,E1 -3128.47,E2 -3128.47} C_VEL
LIN {X 0,Y 552.809,Z 507.853,A -85,B 0,C 180,E1 -3128.953,E2 -3128.953} C_VEL
LIN {X 0,Y 552.627,Z 519.292,A -85,B 0,C 180,E1 -3129.53,E2 -3129.53} C_VEL
LIN {X 0,Y 552.447,Z 531.021,A -85,B 0,C 180,E1 -3130.289,E2 -3130.289} C_VEL
LIN {X 0,Y 552.241,Z 541.731,A -85,B 0,C 180,E1 -3131.16,E2 -3131.16} C_VEL
LIN {X 0,Y 552.082,Z 551.997,A -85,B 0,C 180,E1 -3132.211,E2 -3132.211} C_VEL
LIN {X 0,Y 551.934,Z 560.938,A -85,B 0,C 180,E1 -3133.352,E2 -3133.352} C_VEL
LIN {X 0,Y 551.843,Z 568.004,A -85,B 0,C 180,E1 -3134.488,E2 -3134.488} C_VEL
LIN {X 0,Y 551.775,Z 574.108,A -85,B 0,C 180,E1 -3135.732,E2 -3135.732} C_VEL
LIN {X 0,Y 551.728,Z 577.96,A -85,B 0,C 180,E1 -3136.745,E2 -3136.745} C_VEL
LIN {X 0,Y 551.707,Z 580.251,A -85,B 0,C 180,E1 -3137.493,E2 -3137.493} C_VEL
LIN {X 0,Y 551.713,Z 583.076,A -85,B 0,C 180,E1 -3138.776,E2 -3138.776} C_VEL
LIN {X 0,Y 551.676,Z 584.339,A -85,B 0,C 180,E1 -3139.727,E2 -3139.727} C_VEL
LIN {X 0,Y 551.659,Z 584.876,A -85,B 0,C 180,E1 -3140.467,E2 -3140.467} C_VEL
LIN {X 0,Y 551.671,Z 584.972,A -85,B 0,C 180,E1 -3141.207,E2 -3141.207} C_VEL
LIN {X 0,Y 551.697,Z 584.674,A -85,B 0,C 180,E1 -3141.945,E2 -3141.945} C_VEL
LIN {X 0,Y 551.693,Z 583.99,A -85,B 0,C 180,E1 -3142.681,E2 -3142.681} C_VEL
LIN {X 0,Y 551.734,Z 582.733,A -85,B 0,C 180,E1 -3143.502,E2 -3143.502} C_VEL
LIN {X 0,Y 551.711,Z 579.413,A -85,B 0,C 180,E1 -3144.884,E2 -3144.884} C_VEL
LIN {X 0,Y 551.777,Z 575.638,A -85,B 0,C 180,E1 -3145.983,E2 -3145.983} C_VEL
LIN {X 0,Y 551.779,Z 570.76,A -85,B 0,C 180,E1 -3147.08,E2 -3147.08} C_VEL
LIN {X 0,Y 551.864,Z 564.634,A -85,B 0,C 180,E1 -3148.176,E2 -3148.176} C_VEL
LIN {X 0,Y 552.009,Z 557.034,A -85,B 0,C 180,E1 -3149.271,E2 -3149.271} C_VEL
LIN {X 0,Y 552.136,Z 547.529,A -85,B 0,C 180,E1 -3150.365,E2 -3150.365} C_VEL
LIN {X 0,Y 552.32,Z 537.753,A -85,B 0,C 180,E1 -3151.276,E2 -3151.276} C_VEL
LIN {X 0,Y 552.465,Z 526.824,A -85,B 0,C 180,E1 -3152.096,E2 -3152.096} C_VEL
LIN {X 0,Y 552.675,Z 514.414,A -85,B 0,C 180,E1 -3152.824,E2 -3152.824} C_VEL
LIN {X 0,Y 552.827,Z 502.2,A -85,B 0,C 180,E1 -3153.371,E2 -3153.371} C_VEL
LIN {X 0,Y 552.985,Z 489.223,A -85,B 0,C 180,E1 -3153.78,E2 -3153.78} C_VEL
LIN {X 0,Y 553.135,Z 476.746,A -85,B 0,C 180,E1 -3154.03,E2 -3154.03} C_VEL
LIN {X 0,Y 553.262,Z 380.969,A -85,B 0,C 180,E1 -3155.284,E2 -3155.284} C_VEL
LIN {X 0,Y 552.234,Z 374.587,A -85,B 0,C 180,E1 -3155.408,E2 -3155.408} C_VEL
LIN {X 0,Y 552.374,Z 359.298,A -85,B 0,C 180,E1 -3158.413,E2 -3158.413} C_VEL
LIN {X 0,Y 552.317,Z 353.727,A -85,B 0,C 180,E1 -3159.521,E2 -3159.521} C_VEL
LIN {X 0,Y 552.146,Z 352.709,A -85,B 0,C 180,E1 -3159.756,E2 -3159.756} C_VEL
LIN {X 0,Y 552.154,Z 352.711,A -85,B 0,C 180,E1 -3162.496,E2 -3162.496} C_VEL
LIN {X 0,Y 552.114,Z 352.706,A -85,B 0,C 180,E1 -3165.504,E2 -3165.504} C_VEL
LIN {X 0,Y 552.115,Z 352.708,A -85,B 0,C 180,E1 -3167.788,E2 -3167.788} C_VEL
LIN {X 0,Y 552.132,Z 352.71,A -85,B 0,C 180,E1 -3170.101,E2 -3170.101} C_VEL
LIN {X 0,Y 552.1,Z 352.714,A -85,B 0,C 180,E1 -3172.45,E2 -3172.45} C_VEL
LIN {X 0,Y 552.159,Z 352.701,A -85,B 0,C 180,E1 -3175.35,E2 -3175.35} C_VEL
LIN {X 0,Y 552.129,Z 352.712,A -85,B 0,C 180,E1 -3178.097,E2 -3178.097} C_VEL
LIN {X 0,Y 552.112,Z 352.709,A -85,B 0,C 180,E1 -3180.608,E2 -3180.608} C_VEL
LIN {X 0,Y 552.124,Z 352.705,A -85,B 0,C 180,E1 -3183.184,E2 -3183.184} C_VEL
LIN {X 0,Y 552.115,Z 352.713,A -85,B 0,C 180,E1 -3185.841,E2 -3185.841} C_VEL
LIN {X 0,Y 552.125,Z 352.705,A -85,B 0,C 180,E1 -3189.061,E2 -3189.061} C_VEL
LIN {X 0,Y 552.127,Z 352.708,A -85,B 0,C 180,E1 -3191.444,E2 -3191.444} C_VEL
LIN {X 0,Y 552.093,Z 352.71,A -85,B 0,C 180,E1 -3194.531,E2 -3194.531} C_VEL
LIN {X 0,Y 552.128,Z 352.711,A -85,B 0,C 180,E1 -3197.583,E2 -3197.583} C_VEL
LIN {X 0,Y 552.13,Z 352.706,A -85,B 0,C 180,E1 -3200.472,E2 -3200.472} C_VEL
LIN {X 0,Y 552.107,Z 352.712,A -85,B 0,C 180,E1 -3203.315,E2 -3203.315} C_VEL
LIN {X 0,Y 552.123,Z 352.711,A -85,B 0,C 180,E1 -3205.938,E2 -3205.938} C_VEL
LIN {X 0,Y 552.113,Z 352.707,A -85,B 0,C 180,E1 -3208.54,E2 -3208.54} C_VEL
LIN {X 0,Y 552.12,Z 352.713,A -85,B 0,C 180,E1 -3211.436,E2 -3211.436} C_VEL
LIN {X 0,Y 552.13,Z 352.705,A -85,B 0,C 180,E1 -3214.355,E2 -3214.355} C_VEL
LIN {X 0,Y 552.133,Z 352.706,A -85,B 0,C 180,E1 -3216.759,E2 -3216.759} C_VEL
LIN {X 0,Y 552.121,Z 352.712,A -85,B 0,C 180,E1 -3219.119,E2 -3219.119} C_VEL
LIN {X 0,Y 552.125,Z 352.713,A -85,B 0,C 180,E1 -3221.444,E2 -3221.444} C_VEL
LIN {X 0,Y 552.115,Z 352.71,A -85,B 0,C 180,E1 -3223.737,E2 -3223.737} C_VEL
LIN {X 0,Y 552.129,Z 352.706,A -85,B 0,C 180,E1 -3226.004,E2 -3226.004} C_VEL
LIN {X 0,Y 552.171,Z 352.706,A -85,B 0,C 180,E1 -3228.993,E2 -3228.993} C_VEL
LIN {X 0,Y 552.158,Z 352.702,A -85,B 0,C 180,E1 -3231.951,E2 -3231.951} C_VEL
LIN {X 0,Y 552.227,Z 352.699,A -85,B 0,C 180,E1 -3234.889,E2 -3234.889} C_VEL
LIN {X 0,Y 552.216,Z 352.695,A -85,B 0,C 180,E1 -3237.812,E2 -3237.812} C_VEL
LIN {X 0,Y 552.241,Z 352.697,A -85,B 0,C 180,E1 -3240.729,E2 -3240.729} C_VEL
LIN {X 0,Y 552.205,Z 352.703,A -85,B 0,C 180,E1 -3242.918,E2 -3242.918} C_VEL
LIN {X 0,Y 552.193,Z 352.697,A -85,B 0,C 180,E1 -3245.844,E2 -3245.844} C_VEL
LIN {X 0,Y 552.164,Z 352.708,A -85,B 0,C 180,E1 -3248.785,E2 -3248.785} C_VEL
LIN {X 0,Y 552.155,Z 352.702,A -85,B 0,C 180,E1 -3251.751,E2 -3251.751} C_VEL
LIN {X 0,Y 552.127,Z 352.713,A -85,B 0,C 180,E1 -3254.749,E2 -3254.749} C_VEL
LIN {X 0,Y 552.108,Z 352.708,A -85,B 0,C 180,E1 -3257.789,E2 -3257.789} C_VEL
LIN {X 0,Y 552.126,Z 352.708,A -85,B 0,C 180,E1 -3260.101,E2 -3260.101} C_VEL
LIN {X 0,Y 552.107,Z 352.715,A -85,B 0,C 180,E1 -3262.45,E2 -3262.45} C_VEL
LIN {X 0,Y 552.148,Z 352.703,A -85,B 0,C 180,E1 -3265.351,E2 -3265.351} C_VEL
LIN {X 0,Y 552.119,Z 352.71,A -85,B 0,C 180,E1 -3268.098,E2 -3268.098} C_VEL
LIN {X 0,Y 552.101,Z 352.715,A -85,B 0,C 180,E1 -3270.609,E2 -3270.609} C_VEL
LIN {X 0,Y 552.122,Z 352.706,A -85,B 0,C 180,E1 -3273.185,E2 -3273.185} C_VEL
LIN {X 0,Y 552.106,Z 352.71,A -85,B 0,C 180,E1 -3275.842,E2 -3275.842} C_VEL
LIN {X 0,Y 552.12,Z 352.706,A -85,B 0,C 180,E1 -3279.063,E2 -3279.063} C_VEL
LIN {X 0,Y 552.135,Z 352.704,A -85,B 0,C 180,E1 -3281.445,E2 -3281.445} C_VEL
LIN {X 0,Y 552.092,Z 352.714,A -85,B 0,C 180,E1 -3284.533,E2 -3284.533} C_VEL
LIN {X 0,Y 552.127,Z 352.707,A -85,B 0,C 180,E1 -3287.585,E2 -3287.585} C_VEL
LIN {X 0,Y 552.132,Z 352.708,A -85,B 0,C 180,E1 -3290.474,E2 -3290.474} C_VEL
LIN {X 0,Y 552.113,Z 352.707,A -85,B 0,C 180,E1 -3293.316,E2 -3293.316} C_VEL
LIN {X 0,Y 552.131,Z 352.713,A -85,B 0,C 180,E1 -3295.94,E2 -3295.94} C_VEL
LIN {X 0,Y 552.118,Z 352.707,A -85,B 0,C 180,E1 -3298.541,E2 -3298.541} C_VEL
LIN {X 0,Y 552.126,Z 352.708,A -85,B 0,C 180,E1 -3301.438,E2 -3301.438} C_VEL
LIN {X 0,Y 552.131,Z 352.71,A -85,B 0,C 180,E1 -3304.356,E2 -3304.356} C_VEL
LIN {X 0,Y 552.186,Z 352.885,A -85,B 0,C 180,E1 -3305.617,E2 -3305.617} C_VEL
LIN {X 0,Y 553.294,Z 358.788,A -85,B 0,C 180,E1 -3306.526,E2 -3306.526} C_VEL
LIN {X 0,Y 553.061,Z 376.971,A -85,B 0,C 180,E1 -3309.158,E2 -3309.158} C_VEL
LIN {X 0,Y 552.735,Z 397.214,A -85,B 0,C 180,E1 -3312.041,E2 -3312.041} C_VEL
LIN {X 0,Y 552.475,Z 417.555,A -85,B 0,C 180,E1 -3314.922,E2 -3314.922} C_VEL
LIN {X 0,Y 552.434,Z 422.524,A -85,B 0,C 180,E1 -3315.625,E2 -3315.625} C_VEL
LIN {X 0,Y 553.449,Z 430.323,A -85,B 0,C 180,E1 -3315.757,E2 -3315.757} C_VEL
LIN {X 0,Y 553.15,Z 530.961,A -85,B 0,C 180,E1 -3317.084,E2 -3317.084} C_VEL
LIN {X 0,Y 552.993,Z 543.465,A -85,B 0,C 180,E1 -3317.383,E2 -3317.383} C_VEL
LIN {X 0,Y 552.835,Z 556.377,A -85,B 0,C 180,E1 -3317.846,E2 -3317.846} C_VEL
LIN {X 0,Y 552.626,Z 568.321,A -85,B 0,C 180,E1 -3318.428,E2 -3318.428} C_VEL
LIN {X 0,Y 552.476,Z 580.199,A -85,B 0,C 180,E1 -3319.186,E2 -3319.186} C_VEL
LIN {X 0,Y 552.299,Z 590.607,A -85,B 0,C 180,E1 -3320.016,E2 -3320.016} C_VEL
LIN {X 0,Y 552.125,Z 599.115,A -85,B 0,C 180,E1 -3320.845,E2 -3320.845} C_VEL
LIN {X 0,Y 552.013,Z 606.962,A -85,B 0,C 180,E1 -3321.765,E2 -3321.765} C_VEL
LIN {X 0,Y 551.889,Z 614.623,A -85,B 0,C 180,E1 -3322.868,E2 -3322.868} C_VEL
LIN {X 0,Y 551.867,Z 621.68,A -85,B 0,C 180,E1 -3324.153,E2 -3324.153} C_VEL
LIN {X 0,Y 551.725,Z 626.373,A -85,B 0,C 180,E1 -3325.251,E2 -3325.251} C_VEL
LIN {X 0,Y 551.75,Z 629.958,A -85,B 0,C 180,E1 -3326.349,E2 -3326.349} C_VEL
LIN {X 0,Y 551.723,Z 631.807,A -85,B 0,C 180,E1 -3327.079,E2 -3327.079} C_VEL
LIN {X 0,Y 551.645,Z 634.184,A -85,B 0,C 180,E1 -3328.54,E2 -3328.54} C_VEL
LIN {X 0,Y 551.64,Z 635,A -85,B 0,C 180,E1 -3330,E2 -3330} C_VEL
LIN {X 0,Y 551.645,Z 634.185,A -85,B 0,C 180,E1 -3331.46,E2 -3331.46} C_VEL
LIN {X 0,Y 551.723,Z 631.81,A -85,B 0,C 180,E1 -3332.921,E2 -3332.921} C_VEL
LIN {X 0,Y 551.763,Z 628.896,A -85,B 0,C 180,E1 -3334.017,E2 -3334.017} C_VEL
LIN {X 0,Y 551.724,Z 624.949,A -85,B 0,C 180,E1 -3335.116,E2 -3335.116} C_VEL
LIN {X 0,Y 551.815,Z 619.124,A -85,B 0,C 180,E1 -3336.353,E2 -3336.353} C_VEL
LIN {X 0,Y 551.926,Z 612.237,A -85,B 0,C 180,E1 -3337.499,E2 -3337.499} C_VEL
LIN {X 0,Y 552.082,Z 603.993,A -85,B 0,C 180,E1 -3338.602,E2 -3338.602} C_VEL
LIN {X 0,Y 552.221,Z 595.542,A -85,B 0,C 180,E1 -3339.523,E2 -3339.523} C_VEL
LIN {X 0,Y 552.432,Z 585.096,A -85,B 0,C 180,E1 -3340.445,E2 -3340.445} C_VEL
LIN {X 0,Y 552.555,Z 574.29,A -85,B 0,C 180,E1 -3341.214,E2 -3341.214} C_VEL
LIN {X 0,Y 552.781,Z 563.411,A -85,B 0,C 180,E1 -3341.83,E2 -3341.83} C_VEL
LIN {X 0,Y 552.884,Z 551.772,A -85,B 0,C 180,E1 -3342.34,E2 -3342.34} C_VEL
LIN {X 0,Y 553.047,Z 538.357,A -85,B 0,C 180,E1 -3342.756,E2 -3342.756} C_VEL
LIN {X 0,Y 553.206,Z 525.105,A -85,B 0,C 180,E1 -3343.009,E2 -3343.009} C_VEL
LIN {X 0,Y 553.393,Z 428.984,A -85,B 0,C 180,E1 -3344.262,E2 -3344.262} C_VEL
LIN {X 0,Y 552.427,Z 422.441,A -85,B 0,C 180,E1 -3344.387,E2 -3344.387} C_VEL
LIN {X 0,Y 552.704,Z 400.385,A -85,B 0,C 180,E1 -3347.507,E2 -3347.507} C_VEL
LIN {X 0,Y 552.974,Z 380.942,A -85,B 0,C 180,E1 -3350.263,E2 -3350.263} C_VEL
LIN {X 0,Y 553.347,Z 360.631,A -85,B 0,C 180,E1 -3353.186,E2 -3353.186} C_VEL
LIN {X 0,Y 552.644,Z 355.202,A -85,B 0,C 180,E1 -3354.012,E2 -3354.012} C_VEL
LIN {X 0,Y 552.157,Z 352.71,A -85,B 0,C 180,E1 -3354.435,E2 -3354.435} C_VEL
LIN {X 0,Y 552.144,Z 352.705,A -85,B 0,C 180,E1 -3357.272,E2 -3357.272} C_VEL
LIN {X 0,Y 552.143,Z 352.711,A -85,B 0,C 180,E1 -3360.055,E2 -3360.055} C_VEL
LIN {X 0,Y 552.128,Z 352.705,A -85,B 0,C 180,E1 -3362.848,E2 -3362.848} C_VEL
LIN {X 0,Y 552.107,Z 352.71,A -85,B 0,C 180,E1 -3365.444,E2 -3365.444} C_VEL
LIN {X 0,Y 552.096,Z 352.717,A -85,B 0,C 180,E1 -3367.885,E2 -3367.885} C_VEL
LIN {X 0,Y 552.119,Z 352.706,A -85,B 0,C 180,E1 -3370.479,E2 -3370.479} C_VEL
LIN {X 0,Y 552.098,Z 352.712,A -85,B 0,C 180,E1 -3373.482,E2 -3373.482} C_VEL
LIN {X 0,Y 552.115,Z 352.705,A -85,B 0,C 180,E1 -3376.577,E2 -3376.577} C_VEL
LIN {X 0,Y 552.137,Z 352.709,A -85,B 0,C 180,E1 -3379.521,E2 -3379.521} C_VEL
LIN {X 0,Y 552.088,Z 352.709,A -85,B 0,C 180,E1 -3382.336,E2 -3382.336} C_VEL
LIN {X 0,Y 552.123,Z 352.707,A -85,B 0,C 180,E1 -3385.054,E2 -3385.054} C_VEL
LIN {X 0,Y 552.122,Z 352.712,A -85,B 0,C 180,E1 -3387.682,E2 -3387.682} C_VEL
LIN {X 0,Y 552.138,Z 352.703,A -85,B 0,C 180,E1 -3390.237,E2 -3390.237} C_VEL
LIN {X 0,Y 552.14,Z 352.706,A -85,B 0,C 180,E1 -3392.997,E2 -3392.997} C_VEL
LIN {X 0,Y 552.107,Z 352.71,A -85,B 0,C 180,E1 -3395.161,E2 -3395.161} C_VEL
LIN {X 0,Y 552.107,Z 352.713,A -85,B 0,C 180,E1 -3397.55,E2 -3397.55} C_VEL
LIN {X 0,Y 552.149,Z 352.703,A -85,B 0,C 180,E1 -3400.674,E2 -3400.674} C_VEL
LIN {X 0,Y 552.114,Z 352.707,A -85,B 0,C 180,E1 -3403.737,E2 -3403.737} C_VEL
LIN {X 0,Y 552.129,Z 352.704,A -85,B 0,C 180,E1 -3406.004,E2 -3406.004} C_VEL
LIN {X 0,Y 552.185,Z 352.705,A -85,B 0,C 180,E1 -3408.994,E2 -3408.994} C_VEL
LIN {X 0,Y 552.158,Z 352.701,A -85,B 0,C 180,E1 -3411.952,E2 -3411.952} C_VEL
LIN {X 0,Y 552.227,Z 352.699,A -85,B 0,C 180,E1 -3414.889,E2 -3414.889} C_VEL
LIN {X 0,Y 552.216,Z 352.693,A -85,B 0,C 180,E1 -3417.812,E2 -3417.812} C_VEL
LIN {X 0,Y 552.241,Z 352.697,A -85,B 0,C 180,E1 -3420.729,E2 -3420.729} C_VEL
LIN {X 0,Y 552.205,Z 352.701,A -85,B 0,C 180,E1 -3422.918,E2 -3422.918} C_VEL
LIN {X 0,Y 552.193,Z 352.696,A -85,B 0,C 180,E1 -3425.844,E2 -3425.844} C_VEL
LIN {X 0,Y 552.164,Z 352.708,A -85,B 0,C 180,E1 -3428.786,E2 -3428.786} C_VEL
LIN {X 0,Y 552.156,Z 352.701,A -85,B 0,C 180,E1 -3431.751,E2 -3431.751} C_VEL
LIN {X 0,Y 552.128,Z 352.711,A -85,B 0,C 180,E1 -3434.749,E2 -3434.749} C_VEL
LIN {X 0,Y 552.107,Z 352.707,A -85,B 0,C 180,E1 -3437.789,E2 -3437.789} C_VEL
LIN {X 0,Y 552.127,Z 352.709,A -85,B 0,C 180,E1 -3440.102,E2 -3440.102} C_VEL
LIN {X 0,Y 552.089,Z 352.718,A -85,B 0,C 180,E1 -3442.451,E2 -3442.451} C_VEL
LIN {X 0,Y 552.15,Z 352.699,A -85,B 0,C 180,E1 -3445.352,E2 -3445.352} C_VEL
LIN {X 0,Y 552.12,Z 352.709,A -85,B 0,C 180,E1 -3448.098,E2 -3448.098} C_VEL
LIN {X 0,Y 552.1,Z 352.711,A -85,B 0,C 180,E1 -3450.632,E2 -3450.632} C_VEL
LIN {X 0,Y 552.118,Z 352.706,A -85,B 0,C 180,E1 -3453.186,E2 -3453.186} C_VEL
LIN {X 0,Y 552.11,Z 352.711,A -85,B 0,C 180,E1 -3453.811,E2 -3453.811} C_VEL
LIN {X 0,Y 551.475,Z 352.795,A -85,B 0,C 180,E1 -3454.42,E2 -3454.42} C_VEL
LIN {X 0,Y 548.652,Z 353.146,A -85,B 0,C 180,E1 -3455.408,E2 -3455.408} C_VEL
LIN {X 0,Y 546.23,Z 353.447,A -85,B 0,C 180,E1 -3456.203,E2 -3456.203} C_VEL
LIN {X 0,Y 545.161,Z 353.574,A -85,B 0,C 180,E1 -3456.817,E2 -3456.817} C_VEL
LIN {X 0,Y 545.059,Z 353.585,A -85,B 0,C 180,E1 -3457.025,E2 -3457.025} C_VEL
LIN {X 0,Y 545.09,Z 353.59,A -85,B 0,C 180,E1 -3460.141,E2 -3460.141} C_VEL
LIN {X 0,Y 545.084,Z 353.582,A -85,B 0,C 180,E1 -3463.107,E2 -3463.107} C_VEL
LIN {X 0,Y 545.058,Z 353.591,A -85,B 0,C 180,E1 -3466.226,E2 -3466.226} C_VEL
LIN {X 0,Y 545.101,Z 353.581,A -85,B 0,C 180,E1 -3468.888,E2 -3468.888} C_VEL
LIN {X 0,Y 545.056,Z 353.595,A -85,B 0,C 180,E1 -3471.764,E2 -3471.764} C_VEL
LIN {X 0,Y 545.067,Z 353.586,A -85,B 0,C 180,E1 -3474.535,E2 -3474.535} C_VEL
LIN {X 0,Y 545.083,Z 353.585,A -85,B 0,C 180,E1 -3477.213,E2 -3477.213} C_VEL
LIN {X 0,Y 545.105,Z 353.588,A -85,B 0,C 180,E1 -3479.814,E2 -3479.814} C_VEL
LIN {X 0,Y 545.121,Z 353.614,A -85,B 0,C 180,E1 -3482.242,E2 -3482.242} C_VEL
LIN {X 0,Y 545.441,Z 358.246,A -85,B 0,C 180,E1 -3483.194,E2 -3483.194} C_VEL
LIN {X 0,Y 545.156,Z 373.603,A -85,B 0,C 180,E1 -3486.251,E2 -3486.251} C_VEL
LIN {X 0,Y 545.177,Z 375.099,A -85,B 0,C 180,E1 -3486.508,E2 -3486.508} C_VEL
LIN {X 0,Y 546.569,Z 383.573,A -85,B 0,C 180,E1 -3486.66,E2 -3486.66} C_VEL
LIN {X 0,Y 546.18,Z 481.328,A -85,B 0,C 180,E1 -3487.967,E2 -3487.967} C_VEL
LIN {X 0,Y 546.024,Z 494.877,A -85,B 0,C 180,E1 -3488.307,E2 -3488.307} C_VEL
LIN {X 0,Y 545.879,Z 507.298,A -85,B 0,C 180,E1 -3488.771,E2 -3488.771} C_VEL
LIN {X 0,Y 545.666,Z 518.861,A -85,B 0,C 180,E1 -3489.355,E2 -3489.355} C_VEL
LIN {X 0,Y 545.472,Z 529.695,A -85,B 0,C 180,E1 -3490.053,E2 -3490.053} C_VEL
LIN {X 0,Y 545.254,Z 540.366,A -85,B 0,C 180,E1 -3490.91,E2 -3490.91} C_VEL
LIN {X 0,Y 545.088,Z 549.211,A -85,B 0,C 180,E1 -3491.781,E2 -3491.781} C_VEL
LIN {X 0,Y 544.952,Z 557.288,A -85,B 0,C 180,E1 -3492.746,E2 -3492.746} C_VEL
LIN {X 0,Y 544.791,Z 565.092,A -85,B 0,C 180,E1 -3493.898,E2 -3493.898} C_VEL
LIN {X 0,Y 544.74,Z 571.32,A -85,B 0,C 180,E1 -3495.047,E2 -3495.047} C_VEL
LIN {X 0,Y 544.681,Z 576.204,A -85,B 0,C 180,E1 -3496.19,E2 -3496.19} C_VEL
LIN {X 0,Y 544.624,Z 579.91,A -85,B 0,C 180,E1 -3497.328,E2 -3497.328} C_VEL
LIN {X 0,Y 544.625,Z 583.059,A -85,B 0,C 180,E1 -3498.736,E2 -3498.736} C_VEL
LIN {X 0,Y 544.58,Z 584.211,A -85,B 0,C 180,E1 -3499.591,E2 -3499.591} C_VEL
LIN {X 0,Y 544.582,Z 584.81,A -85,B 0,C 180,E1 -3500.342,E2 -3500.342} C_VEL
LIN {X 0,Y 544.564,Z 584.996,A -85,B 0,C 180,E1 -3501.091,E2 -3501.091} C_VEL
LIN {X 0,Y 544.612,Z 584.75,A -85,B 0,C 180,E1 -3501.839,E2 -3501.839} C_VEL
LIN {X 0,Y 544.653,Z 583.091,A -85,B 0,C 180,E1 -3503.331,E2 -3503.331} C_VEL
LIN {X 0,Y 544.645,Z 581.642,A -85,B 0,C 180,E1 -3504.075,E2 -3504.075} C_VEL
LIN {X 0,Y 544.603,Z 578.669,A -85,B 0,C 180,E1 -3505.188,E2 -3505.188} C_VEL
LIN {X 0,Y 544.693,Z 574.653,A -85,B 0,C 180,E1 -3506.301,E2 -3506.301} C_VEL
LIN {X 0,Y 544.774,Z 568.493,A -85,B 0,C 180,E1 -3507.597,E2 -3507.597} C_VEL
LIN {X 0,Y 544.874,Z 561.81,A -85,B 0,C 180,E1 -3508.707,E2 -3508.707} C_VEL
LIN {X 0,Y 544.993,Z 553.548,A -85,B 0,C 180,E1 -3509.815,E2 -3509.815} C_VEL
LIN {X 0,Y 545.153,Z 545.071,A -85,B 0,C 180,E1 -3510.739,E2 -3510.739} C_VEL
LIN {X 0,Y 545.354,Z 534.658,A -85,B 0,C 180,E1 -3511.662,E2 -3511.662} C_VEL
LIN {X 0,Y 545.553,Z 522.962,A -85,B 0,C 180,E1 -3512.492,E2 -3512.492} C_VEL
LIN {X 0,Y 545.786,Z 511.207,A -85,B 0,C 180,E1 -3513.137,E2 -3513.137} C_VEL
LIN {X 0,Y 545.937,Z 499.076,A -85,B 0,C 180,E1 -3513.644,E2 -3513.644} C_VEL
LIN {X 0,Y 546.082,Z 486.626,A -85,B 0,C 180,E1 -3514.013,E2 -3514.013} C_VEL
LIN {X 0,Y 546.212,Z 471.97,A -85,B 0,C 180,E1 -3514.266,E2 -3514.266} C_VEL
LIN {X 0,Y 546.416,Z 381.943,A -85,B 0,C 180,E1 -3515.456,E2 -3515.456} C_VEL
LIN {X 0,Y 545.238,Z 374.852,A -85,B 0,C 180,E1 -3515.594,E2 -3515.594} C_VEL
LIN {X 0,Y 545.457,Z 358.277,A -85,B 0,C 180,E1 -3518.894,E2 -3518.894} C_VEL
LIN {X 0,Y 545.097,Z 353.588,A -85,B 0,C 180,E1 -3519.883,E2 -3519.883} C_VEL
LIN {X 0,Y 545.097,Z 353.588,A -85,B 0,C 180,E1 -3522.661,E2 -3522.661} C_VEL
LIN {X 0,Y 545.092,Z 353.583,A -85,B 0,C 180,E1 -3524.943,E2 -3524.943} C_VEL
LIN {X 0,Y 545.083,Z 353.587,A -85,B 0,C 180,E1 -3528.025,E2 -3528.025} C_VEL
LIN {X 0,Y 545.097,Z 353.589,A -85,B 0,C 180,E1 -3530.371,E2 -3530.371} C_VEL
LIN {X 0,Y 545.096,Z 353.582,A -85,B 0,C 180,E1 -3533.558,E2 -3533.558} C_VEL
LIN {X 0,Y 545.083,Z 353.588,A -85,B 0,C 180,E1 -3536,E2 -3536} C_VEL
LIN {X 0,Y 545.095,Z 353.582,A -85,B 0,C 180,E1 -3538.748,E2 -3538.748} C_VEL
LIN {X 0,Y 545.071,Z 353.584,A -85,B 0,C 180,E1 -3541.047,E2 -3541.047} C_VEL
LIN {X 0,Y 545.073,Z 353.588,A -85,B 0,C 180,E1 -3543.67,E2 -3543.67} C_VEL
LIN {X 0,Y 545.057,Z 353.59,A -85,B 0,C 180,E1 -3546.378,E2 -3546.378} C_VEL
LIN {X 0,Y 545.104,Z 353.581,A -85,B 0,C 180,E1 -3549.323,E2 -3549.323} C_VEL
LIN {X 0,Y 545.077,Z 353.59,A -85,B 0,C 180,E1 -3552.102,E2 -3552.102} C_VEL
LIN {X 0,Y 545.061,Z 353.587,A -85,B 0,C 180,E1 -3555.166,E2 -3555.166} C_VEL
LIN {X 0,Y 545.08,Z 353.591,A -85,B 0,C 180,E1 -3557.897,E2 -3557.897} C_VEL
LIN {X 0,Y 545.101,Z 353.581,A -85,B 0,C 180,E1 -3560.675,E2 -3560.675} C_VEL
LIN {X 0,Y 545.046,Z 353.594,A -85,B 0,C 180,E1 -3563.619,E2 -3563.619} C_VEL
LIN {X 0,Y 545.064,Z 353.586,A -85,B 0,C 180,E1 -3566.328,E2 -3566.328} C_VEL
LIN {X 0,Y 545.062,Z 353.587,A -85,B 0,C 180,E1 -3568.951,E2 -3568.951} C_VEL
LIN {X 0,Y 545.099,Z 353.588,A -85,B 0,C 180,E1 -3571.507,E2 -3571.507} C_VEL
LIN {X 0,Y 545.092,Z 353.582,A -85,B 0,C 180,E1 -3574.489,E2 -3574.489} C_VEL
LIN {X 0,Y 545.061,Z 353.592,A -85,B 0,C 180,E1 -3577.243,E2 -3577.243} C_VEL
LIN {X 0,Y 545.113,Z 353.579,A -85,B 0,C 180,E1 -3580.414,E2 -3580.414} C_VEL
LIN {X 0,Y 545.071,Z 353.591,A -85,B 0,C 180,E1 -3583.521,E2 -3583.521} C_VEL
LIN {X 0,Y 545.088,Z 353.585,A -85,B 0,C 180,E1 -3585.819,E2 -3585.819} C_VEL
LIN {X 0,Y 545.124,Z 353.582,A -85,B 0,C 180,E1 -3588.849,E2 -3588.849} C_VEL
LIN {X 0,Y 545.128,Z 353.579,A -85,B 0,C 180,E1 -3591.847,E2 -3591.847} C_VEL
LIN {X 0,Y 545.202,Z 353.574,A -85,B 0,C 180,E1 -3594.823,E2 -3594.823} C_VEL
LIN {X 0,Y 545.188,Z 353.571,A -85,B 0,C 180,E1 -3597.783,E2 -3597.783} C_VEL
LIN {X 0,Y 545.21,Z 353.573,A -85,B 0,C 180,E1 -3600.738,E2 -3600.738} C_VEL
LIN {X 0,Y 545.171,Z 353.579,A -85,B 0,C 180,E1 -3602.956,E2 -3602.956} C_VEL
LIN {X 0,Y 545.164,Z 353.573,A -85,B 0,C 180,E1 -3605.919,E2 -3605.919} C_VEL
LIN {X 0,Y 545.12,Z 353.585,A -85,B 0,C 180,E1 -3608.9,E2 -3608.9} C_VEL
LIN {X 0,Y 545.127,Z 353.578,A -85,B 0,C 180,E1 -3611.904,E2 -3611.904} C_VEL
LIN {X 0,Y 545.077,Z 353.59,A -85,B 0,C 180,E1 -3614.944,E2 -3614.944} C_VEL
LIN {X 0,Y 545.075,Z 353.585,A -85,B 0,C 180,E1 -3618.026,E2 -3618.026} C_VEL
LIN {X 0,Y 545.091,Z 353.587,A -85,B 0,C 180,E1 -3620.372,E2 -3620.372} C_VEL
LIN {X 0,Y 545.106,Z 353.58,A -85,B 0,C 180,E1 -3623.558,E2 -3623.558} C_VEL
LIN {X 0,Y 545.081,Z 353.585,A -85,B 0,C 180,E1 -3626,E2 -3626} C_VEL
LIN {X 0,Y 545.083,Z 353.588,A -85,B 0,C 180,E1 -3628.749,E2 -3628.749} C_VEL
LIN {X 0,Y 545.071,Z 353.585,A -85,B 0,C 180,E1 -3631.683,E2 -3631.683} C_VEL
LIN {X 0,Y 545.077,Z 353.589,A -85,B 0,C 180,E1 -3634.563,E2 -3634.563} C_VEL
LIN {X 0,Y 545.035,Z 353.589,A -85,B 0,C 180,E1 -3637.304,E2 -3637.304} C_VEL
LIN {X 0,Y 545.087,Z 353.59,A -85,B 0,C 180,E1 -3640.141,E2 -3640.141} C_VEL
LIN {X 0,Y 545.082,Z 353.583,A -85,B 0,C 180,E1 -3643.106,E2 -3643.106} C_VEL
LIN {X 0,Y 545.062,Z 353.592,A -85,B 0,C 180,E1 -3646.225,E2 -3646.225} C_VEL
LIN {X 0,Y 545.094,Z 353.581,A -85,B 0,C 180,E1 -3648.888,E2 -3648.888} C_VEL
LIN {X 0,Y 545.052,Z 353.591,A -85,B 0,C 180,E1 -3651.764,E2 -3651.764} C_VEL
LIN {X 0,Y 545.064,Z 353.587,A -85,B 0,C 180,E1 -3654.535,E2 -3654.535} C_VEL
LIN {X 0,Y 545.081,Z 353.583,A -85,B 0,C 180,E1 -3657.213,E2 -3657.213} C_VEL
LIN {X 0,Y 545.102,Z 353.588,A -85,B 0,C 180,E1 -3659.814,E2 -3659.814} C_VEL
LIN {X 0,Y 545.097,Z 353.582,A -85,B 0,C 180,E1 -3662.827,E2 -3662.827} C_VEL
LIN {X 0,Y 545.118,Z 353.628,A -85,B 0,C 180,E1 -3665.432,E2 -3665.432} C_VEL
LIN {X 0,Y 546.377,Z 360.419,A -85,B 0,C 180,E1 -3666.501,E2 -3666.501} C_VEL
LIN {X 0,Y 546.079,Z 379.396,A -85,B 0,C 180,E1 -3669.273,E2 -3669.273} C_VEL
LIN {X 0,Y 545.723,Z 400.02,A -85,B 0,C 180,E1 -3672.242,E2 -3672.242} C_VEL
LIN {X 0,Y 545.443,Z 422.697,A -85,B 0,C 180,E1 -3675.444,E2 -3675.444} C_VEL
LIN {X 0,Y 546.578,Z 430.527,A -85,B 0,C 180,E1 -3675.578,E2 -3675.578} C_VEL
LIN {X 0,Y 546.254,Z 530.961,A -85,B 0,C 180,E1 -3676.918,E2 -3676.918} C_VEL
LIN {X 0,Y 546.061,Z 544.226,A -85,B 0,C 180,E1 -3677.244,E2 -3677.244} C_VEL
LIN {X 0,Y 545.891,Z 556.375,A -85,B 0,C 180,E1 -3677.688,E2 -3677.688} C_VEL
LIN {X 0,Y 545.699,Z 567.471,A -85,B 0,C 180,E1 -3678.231,E2 -3678.231} C_VEL
LIN {X 0,Y 545.525,Z 578.906,A -85,B 0,C 180,E1 -3678.952,E2 -3678.952} C_VEL
LIN {X 0,Y 545.286,Z 589.539,A -85,B 0,C 180,E1 -3679.792,E2 -3679.792} C_VEL
LIN {X 0,Y 545.084,Z 599.115,A -85,B 0,C 180,E1 -3680.726,E2 -3680.726} C_VEL
LIN {X 0,Y 544.977,Z 606.962,A -85,B 0,C 180,E1 -3681.658,E2 -3681.658} C_VEL
LIN {X 0,Y 544.823,Z 614.622,A -85,B 0,C 180,E1 -3682.775,E2 -3682.775} C_VEL
LIN {X 0,Y 544.776,Z 621.68,A -85,B 0,C 180,E1 -3684.076,E2 -3684.076} C_VEL
LIN {X 0,Y 544.629,Z 626.373,A -85,B 0,C 180,E1 -3685.189,E2 -3685.189} C_VEL
LIN {X 0,Y 544.669,Z 629.958,A -85,B 0,C 180,E1 -3686.301,E2 -3686.301} C_VEL
LIN {X 0,Y 544.65,Z 631.807,A -85,B 0,C 180,E1 -3687.041,E2 -3687.041} C_VEL
LIN {X 0,Y 544.546,Z 634.183,A -85,B 0,C 180,E1 -3688.521,E2 -3688.521} C_VEL
LIN {X 0,Y 544.541,Z 635,A -85,B 0,C 180,E1 -3690,E2 -3690} C_VEL
LIN {X 0,Y 544.546,Z 634.184,A -85,B 0,C 180,E1 -3691.479,E2 -3691.479} C_VEL
LIN {X 0,Y 544.65,Z 631.81,A -85,B 0,C 180,E1 -3692.959,E2 -3692.959} C_VEL
LIN {X 0,Y 544.683,Z 628.896,A -85,B 0,C 180,E1 -3694.069,E2 -3694.069} C_VEL
LIN {X 0,Y 544.654,Z 624.949,A -85,B 0,C 180,E1 -3695.182,E2 -3695.182} C_VEL
LIN {X 0,Y 544.729,Z 619.643,A -85,B 0,C 180,E1 -3696.34,E2 -3696.34} C_VEL
LIN {X 0,Y 544.836,Z 613.468,A -85,B 0,C 180,E1 -3697.411,E2 -3697.411} C_VEL
LIN {X 0,Y 545.006,Z 605.479,A -85,B 0,C 180,E1 -3698.528,E2 -3698.528} C_VEL
LIN {X 0,Y 545.152,Z 597.335,A -85,B 0,C 180,E1 -3699.46,E2 -3699.46} C_VEL
LIN {X 0,Y 545.376,Z 587.4,A -85,B 0,C 180,E1 -3700.393,E2 -3700.393} C_VEL
LIN {X 0,Y 545.569,Z 576.596,A -85,B 0,C 180,E1 -3701.207,E2 -3701.207} C_VEL
LIN {X 0,Y 545.746,Z 565.176,A -85,B 0,C 180,E1 -3701.89,E2 -3701.89} C_VEL
LIN {X 0,Y 545.93,Z 552.979,A -85,B 0,C 180,E1 -3702.452,E2 -3702.452} C_VEL
LIN {X 0,Y 546.121,Z 540.184,A -85,B 0,C 180,E1 -3702.873,E2 -3702.873} C_VEL
LIN {X 0,Y 546.297,Z 526.619,A -85,B 0,C 180,E1 -3703.152,E2 -3703.152} C_VEL
LIN {X 0,Y 546.457,Z 429.559,A -85,B 0,C 180,E1 -3704.438,E2 -3704.438} C_VEL
LIN {X 0,Y 545.439,Z 422.471,A -85,B 0,C 180,E1 -3704.561,E2 -3704.561} C_VEL
LIN {X 0,Y 545.696,Z 399.958,A -85,B 0,C 180,E1 -3707.757,E2 -3707.757} C_VEL
LIN {X 0,Y 545.989,Z 381.992,A -85,B 0,C 180,E1 -3710.337,E2 -3710.337} C_VEL
LIN {X 0,Y 546.422,Z 361.718,A -85,B 0,C 180,E1 -3713.297,E2 -3713.297} C_VEL
LIN {X 0,Y 545.385,Z 354.921,A -85,B 0,C 180,E1 -3714.353,E2 -3714.353} C_VEL
LIN {X 0,Y 545.108,Z 353.586,A -85,B 0,C 180,E1 -3714.569,E2 -3714.569} C_VEL
LIN {X 0,Y 545.094,Z 353.586,A -85,B 0,C 180,E1 -3717.655,E2 -3717.655} C_VEL
LIN {X 0,Y 545.096,Z 353.586,A -85,B 0,C 180,E1 -3720.249,E2 -3720.249} C_VEL
LIN {X 0,Y 545.088,Z 353.582,A -85,B 0,C 180,E1 -3723.063,E2 -3723.063} C_VEL
LIN {X 0,Y 545.062,Z 353.591,A -85,B 0,C 180,E1 -3725.677,E2 -3725.677} C_VEL
LIN {X 0,Y 545.052,Z 353.59,A -85,B 0,C 180,E1 -3728.236,E2 -3728.236} C_VEL
LIN {X 0,Y 545.094,Z 353.581,A -85,B 0,C 180,E1 -3731.112,E2 -3731.112} C_VEL
LIN {X 0,Y 545.05,Z 353.589,A -85,B 0,C 180,E1 -3734.129,E2 -3734.129} C_VEL
LIN {X 0,Y 545.082,Z 353.581,A -85,B 0,C 180,E1 -3736.894,E2 -3736.894} C_VEL
LIN {X 0,Y 545.087,Z 353.587,A -85,B 0,C 180,E1 -3739.859,E2 -3739.859} C_VEL
LIN {X 0,Y 545.073,Z 353.585,A -85,B 0,C 180,E1 -3743.072,E2 -3743.072} C_VEL
LIN {X 0,Y 545.083,Z 353.591,A -85,B 0,C 180,E1 -3745.605,E2 -3745.605} C_VEL
LIN {X 0,Y 545.071,Z 353.584,A -85,B 0,C 180,E1 -3748.317,E2 -3748.317} C_VEL
LIN {X 0,Y 545.086,Z 353.588,A -85,B 0,C 180,E1 -3751.25,E2 -3751.25} C_VEL
LIN {X 0,Y 545.081,Z 353.58,A -85,B 0,C 180,E1 -3754,E2 -3754} C_VEL
LIN {X 0,Y 545.106,Z 353.576,A -85,B 0,C 180,E1 -3756.442,E2 -3756.442} C_VEL
LIN {X 0,Y 545.091,Z 353.584,A -85,B 0,C 180,E1 -3759.628,E2 -3759.628} C_VEL
LIN {X 0,Y 545.088,Z 353.584,A -85,B 0,C 180,E1 -3762.75,E2 -3762.75} C_VEL
LIN {X 0,Y 545.087,Z 353.582,A -85,B 0,C 180,E1 -3765.82,E2 -3765.82} C_VEL
LIN {X 0,Y 545.135,Z 353.581,A -85,B 0,C 180,E1 -3768.85,E2 -3768.85} C_VEL
LIN {X 0,Y 545.128,Z 353.577,A -85,B 0,C 180,E1 -3771.847,E2 -3771.847} C_VEL
LIN {X 0,Y 545.201,Z 353.573,A -85,B 0,C 180,E1 -3774.823,E2 -3774.823} C_VEL
LIN {X 0,Y 545.187,Z 353.568,A -85,B 0,C 180,E1 -3777.784,E2 -3777.784} C_VEL
LIN {X 0,Y 545.211,Z 353.573,A -85,B 0,C 180,E1 -3780.739,E2 -3780.739} C_VEL
LIN {X 0,Y 545.171,Z 353.576,A -85,B 0,C 180,E1 -3782.956,E2 -3782.956} C_VEL
LIN {X 0,Y 545.164,Z 353.572,A -85,B 0,C 180,E1 -3785.92,E2 -3785.92} C_VEL
LIN {X 0,Y 545.12,Z 353.583,A -85,B 0,C 180,E1 -3788.9,E2 -3788.9} C_VEL
LIN {X 0,Y 545.127,Z 353.577,A -85,B 0,C 180,E1 -3791.905,E2 -3791.905} C_VEL
LIN {X 0,Y 545.077,Z 353.586,A -85,B 0,C 180,E1 -3794.944,E2 -3794.944} C_VEL
LIN {X 0,Y 545.075,Z 353.585,A -85,B 0,C 180,E1 -3798.026,E2 -3798.026} C_VEL
LIN {X 0,Y 545.091,Z 353.589,A -85,B 0,C 180,E1 -3800.373,E2 -3800.373} C_VEL
LIN {X 0,Y 545.084,Z 353.582,A -85,B 0,C 180,E1 -3803.56,E2 -3803.56} C_VEL
LIN {X 0,Y 545.082,Z 353.584,A -85,B 0,C 180,E1 -3806.001,E2 -3806.001} C_VEL
LIN {X 0,Y 545.084,Z 353.585,A -85,B 0,C 180,E1 -3808.749,E2 -3808.749} C_VEL
LIN {X 0,Y 545.073,Z 353.584,A -85,B 0,C 180,E1 -3811.683,E2 -3811.683} C_VEL
LIN {X 0,Y 545.076,Z 353.587,A -85,B 0,C 180,E1 -3814.564,E2 -3814.564} C_VEL
LIN {X 0,Y 545.059,Z 353.585,A -85,B 0,C 180,E1 -3817.025,E2 -3817.025} C_VEL
LIN {X 0,Y 544.355,Z 353.677,A -85,B 0,C 180,E1 -3817.642,E2 -3817.642} C_VEL
LIN {X 0,Y 541.502,Z 354.03,A -85,B 0,C 180,E1 -3818.643,E2 -3818.643} C_VEL
LIN {X 0,Y 539.125,Z 354.327,A -85,B 0,C 180,E1 -3819.449,E2 -3819.449} C_VEL
LIN {X 0,Y 538.12,Z 354.459,A -85,B 0,C 180,E1 -3820.071,E2 -3820.071} C_VEL
LIN {X 0,Y 538.045,Z 354.46,A -85,B 0,C 180,E1 -3820.281,E2 -3820.281} C_VEL
LIN {X 0,Y 538.03,Z 354.461,A -85,B 0,C 180,E1 -3822.989,E2 -3822.989} C_VEL
LIN {X 0,Y 538.024,Z 354.47,A -85,B 0,C 180,E1 -3825.927,E2 -3825.927} C_VEL
LIN {X 0,Y 538.078,Z 354.458,A -85,B 0,C 180,E1 -3829.25,E2 -3829.25} C_VEL
LIN {X 0,Y 537.995,Z 354.471,A -85,B 0,C 180,E1 -3832.124,E2 -3832.124} C_VEL
LIN {X 0,Y 538.022,Z 354.463,A -85,B 0,C 180,E1 -3834.918,E2 -3834.918} C_VEL
LIN {X 0,Y 538.028,Z 354.47,A -85,B 0,C 180,E1 -3837.619,E2 -3837.619} C_VEL
LIN {X 0,Y 538.046,Z 354.463,A -85,B 0,C 180,E1 -3840.241,E2 -3840.241} C_VEL
LIN {X 0,Y 538.092,Z 354.596,A -85,B 0,C 180,E1 -3842.129,E2 -3842.129} C_VEL
LIN {X 0,Y 538.481,Z 359.939,A -85,B 0,C 180,E1 -3843.239,E2 -3843.239} C_VEL
LIN {X 0,Y 538.152,Z 375.15,A -85,B 0,C 180,E1 -3846.298,E2 -3846.298} C_VEL
LIN {X 0,Y 539.69,Z 384.541,A -85,B 0,C 180,E1 -3846.481,E2 -3846.481} C_VEL
LIN {X 0,Y 539.292,Z 481.576,A -85,B 0,C 180,E1 -3847.795,E2 -3847.795} C_VEL
LIN {X 0,Y 539.126,Z 494.391,A -85,B 0,C 180,E1 -3848.116,E2 -3848.116} C_VEL
LIN {X 0,Y 538.955,Z 507.022,A -85,B 0,C 180,E1 -3848.585,E2 -3848.585} C_VEL
LIN {X 0,Y 538.727,Z 518.75,A -85,B 0,C 180,E1 -3849.177,E2 -3849.177} C_VEL
LIN {X 0,Y 538.534,Z 529.543,A -85,B 0,C 180,E1 -3849.879,E2 -3849.879} C_VEL
LIN {X 0,Y 538.285,Z 540.287,A -85,B 0,C 180,E1 -3850.752,E2 -3850.752} C_VEL
LIN {X 0,Y 538.06,Z 550.016,A -85,B 0,C 180,E1 -3851.731,E2 -3851.731} C_VEL
LIN {X 0,Y 537.836,Z 559.282,A -85,B 0,C 180,E1 -3852.902,E2 -3852.902} C_VEL
LIN {X 0,Y 537.707,Z 566.687,A -85,B 0,C 180,E1 -3854.07,E2 -3854.07} C_VEL
LIN {X 0,Y 537.633,Z 572.931,A -85,B 0,C 180,E1 -3855.317,E2 -3855.317} C_VEL
LIN {X 0,Y 537.577,Z 577.16,A -85,B 0,C 180,E1 -3856.39,E2 -3856.39} C_VEL
LIN {X 0,Y 537.535,Z 579.567,A -85,B 0,C 180,E1 -3857.158,E2 -3857.158} C_VEL
LIN {X 0,Y 537.493,Z 581.526,A -85,B 0,C 180,E1 -3857.924,E2 -3857.924} C_VEL
LIN {X 0,Y 537.543,Z 583.036,A -85,B 0,C 180,E1 -3858.69,E2 -3858.69} C_VEL
LIN {X 0,Y 537.481,Z 584.733,A -85,B 0,C 180,E1 -3860.213,E2 -3860.213} C_VEL
LIN {X 0,Y 537.461,Z 584.991,A -85,B 0,C 180,E1 -3860.972,E2 -3860.972} C_VEL
LIN {X 0,Y 537.508,Z 584.826,A -85,B 0,C 180,E1 -3861.731,E2 -3861.731} C_VEL
LIN {X 0,Y 537.553,Z 583.268,A -85,B 0,C 180,E1 -3863.243,E2 -3863.243} C_VEL
LIN {X 0,Y 537.548,Z 581.902,A -85,B 0,C 180,E1 -3863.996,E2 -3863.996} C_VEL
LIN {X 0,Y 537.516,Z 579.019,A -85,B 0,C 180,E1 -3865.125,E2 -3865.125} C_VEL
LIN {X 0,Y 537.612,Z 575.112,A -85,B 0,C 180,E1 -3866.252,E2 -3866.252} C_VEL
LIN {X 0,Y 537.649,Z 570.093,A -85,B 0,C 180,E1 -3867.378,E2 -3867.378} C_VEL
LIN {X 0,Y 537.751,Z 563.844,A -85,B 0,C 180,E1 -3868.502,E2 -3868.502} C_VEL
LIN {X 0,Y 537.93,Z 556.051,A -85,B 0,C 180,E1 -3869.626,E2 -3869.626} C_VEL
LIN {X 0,Y 538.133,Z 546.389,A -85,B 0,C 180,E1 -3870.748,E2 -3870.748} C_VEL
LIN {X 0,Y 538.342,Z 536.339,A -85,B 0,C 180,E1 -3871.683,E2 -3871.683} C_VEL
LIN {X 0,Y 538.557,Z 525.019,A -85,B 0,C 180,E1 -3872.524,E2 -3872.524} C_VEL
LIN {X 0,Y 538.817,Z 513.885,A -85,B 0,C 180,E1 -3873.178,E2 -3873.178} C_VEL
LIN {X 0,Y 538.968,Z 502.59,A -85,B 0,C 180,E1 -3873.691,E2 -3873.691} C_VEL
LIN {X 0,Y 539.165,Z 489.641,A -85,B 0,C 180,E1 -3874.111,E2 -3874.111} C_VEL
LIN {X 0,Y 539.327,Z 477.196,A -85,B 0,C 180,E1 -3874.367,E2 -3874.367} C_VEL
LIN {X 0,Y 539.618,Z 383.171,A -85,B 0,C 180,E1 -3875.629,E2 -3875.629} C_VEL
LIN {X 0,Y 538.249,Z 375.157,A -85,B 0,C 180,E1 -3875.784,E2 -3875.784} C_VEL
LIN {X 0,Y 538.482,Z 359.136,A -85,B 0,C 180,E1 -3879.01,E2 -3879.01} C_VEL
LIN {X 0,Y 538.034,Z 354.469,A -85,B 0,C 180,E1 -3880.014,E2 -3880.014} C_VEL
LIN {X 0,Y 538.089,Z 354.46,A -85,B 0,C 180,E1 -3882.062,E2 -3882.062} C_VEL
LIN {X 0,Y 538.051,Z 354.458,A -85,B 0,C 180,E1 -3885.143,E2 -3885.143} C_VEL
LIN {X 0,Y 538.035,Z 354.468,A -85,B 0,C 180,E1 -3888.27,E2 -3888.27} C_VEL
LIN {X 0,Y 538.042,Z 354.463,A -85,B 0,C 180,E1 -3890.651,E2 -3890.651} C_VEL
LIN {X 0,Y 538.029,Z 354.465,A -85,B 0,C 180,E1 -3893.887,E2 -3893.887} C_VEL
LIN {X 0,Y 538.046,Z 354.466,A -85,B 0,C 180,E1 -3896.366,E2 -3896.366} C_VEL
LIN {X 0,Y 538.06,Z 354.458,A -85,B 0,C 180,E1 -3898.938,E2 -3898.938} C_VEL
LIN {X 0,Y 538.016,Z 354.469,A -85,B 0,C 180,E1 -3901.887,E2 -3901.887} C_VEL
LIN {X 0,Y 538.033,Z 354.463,A -85,B 0,C 180,E1 -3904.62,E2 -3904.62} C_VEL
LIN {X 0,Y 538.008,Z 354.464,A -85,B 0,C 180,E1 -3907.17,E2 -3907.17} C_VEL
LIN {X 0,Y 538.027,Z 354.468,A -85,B 0,C 180,E1 -3909.795,E2 -3909.795} C_VEL
LIN {X 0,Y 538.016,Z 354.463,A -85,B 0,C 180,E1 -3912.785,E2 -3912.785} C_VEL
LIN {X 0,Y 538.03,Z 354.462,A -85,B 0,C 180,E1 -3915.14,E2 -3915.14} C_VEL
LIN {X 0,Y 538.038,Z 354.464,A -85,B 0,C 180,E1 -3918.227,E2 -3918.227} C_VEL
LIN {X 0,Y 538.055,Z 354.46,A -85,B 0,C 180,E1 -3920.411,E2 -3920.411} C_VEL
LIN {X 0,Y 538.023,Z 354.464,A -85,B 0,C 180,E1 -3923.066,E2 -3923.066} C_VEL
LIN {X 0,Y 538.02,Z 354.47,A -85,B 0,C 180,E1 -3925.826,E2 -3925.826} C_VEL
LIN {X 0,Y 538.018,Z 354.463,A -85,B 0,C 180,E1 -3928.499,E2 -3928.499} C_VEL
LIN {X 0,Y 538.053,Z 354.462,A -85,B 0,C 180,E1 -3931.099,E2 -3931.099} C_VEL
LIN {X 0,Y 538.043,Z 354.467,A -85,B 0,C 180,E1 -3933.633,E2 -3933.633} C_VEL
LIN {X 0,Y 538.034,Z 354.463,A -85,B 0,C 180,E1 -3936.113,E2 -3936.113} C_VEL
LIN {X 0,Y 538.036,Z 354.467,A -85,B 0,C 180,E1 -3939.348,E2 -3939.348} C_VEL
LIN {X 0,Y 538.064,Z 354.458,A -85,B 0,C 180,E1 -3942.517,E2 -3942.517} C_VEL
LIN {X 0,Y 538.056,Z 354.463,A -85,B 0,C 180,E1 -3945.63,E2 -3945.63} C_VEL
LIN {X 0,Y 538.081,Z 354.458,A -85,B 0,C 180,E1 -3948.701,E2 -3948.701} C_VEL
LIN {X 0,Y 538.084,Z 354.457,A -85,B 0,C 180,E1 -3951.739,E2 -3951.739} C_VEL
LIN {X 0,Y 538.158,Z 354.45,A -85,B 0,C 180,E1 -3954.755,E2 -3954.755} C_VEL
LIN {X 0,Y 538.16,Z 354.447,A -85,B 0,C 180,E1 -3957.754,E2 -3957.754} C_VEL
LIN {X 0,Y 538.18,Z 354.449,A -85,B 0,C 180,E1 -3960.748,E2 -3960.748} C_VEL
LIN {X 0,Y 538.137,Z 354.455,A -85,B 0,C 180,E1 -3962.994,E2 -3962.994} C_VEL
LIN {X 0,Y 538.117,Z 354.451,A -85,B 0,C 180,E1 -3965.997,E2 -3965.997} C_VEL
LIN {X 0,Y 538.07,Z 354.463,A -85,B 0,C 180,E1 -3969.017,E2 -3969.017} C_VEL
LIN {X 0,Y 538.075,Z 354.457,A -85,B 0,C 180,E1 -3972.063,E2 -3972.063} C_VEL
LIN {X 0,Y 538.037,Z 354.464,A -85,B 0,C 180,E1 -3975.144,E2 -3975.144} C_VEL
LIN {X 0,Y 538.027,Z 354.466,A -85,B 0,C 180,E1 -3978.27,E2 -3978.27} C_VEL
LIN {X 0,Y 538.035,Z 354.468,A -85,B 0,C 180,E1 -3980.651,E2 -3980.651} C_VEL
LIN {X 0,Y 538.033,Z 354.462,A -85,B 0,C 180,E1 -3983.887,E2 -3983.887} C_VEL
LIN {X 0,Y 538.042,Z 354.467,A -85,B 0,C 180,E1 -3986.367,E2 -3986.367} C_VEL
LIN {X 0,Y 538.024,Z 354.465,A -85,B 0,C 180,E1 -3988.934,E2 -3988.934} C_VEL
LIN {X 0,Y 538.021,Z 354.465,A -85,B 0,C 180,E1 -3991.891,E2 -3991.891} C_VEL
LIN {X 0,Y 538.027,Z 354.467,A -85,B 0,C 180,E1 -3994.622,E2 -3994.622} C_VEL
LIN {X 0,Y 538.004,Z 354.465,A -85,B 0,C 180,E1 -3997.172,E2 -3997.172} C_VEL
LIN {X 0,Y 538.048,Z 354.462,A -85,B 0,C 180,E1 -3999.795,E2 -3999.795} C_VEL
LIN {X 0,Y 538.019,Z 354.465,A -85,B 0,C 180,E1 -4002.786,E2 -4002.786} C_VEL
LIN {X 0,Y 538.025,Z 354.467,A -85,B 0,C 180,E1 -4005.926,E2 -4005.926} C_VEL
LIN {X 0,Y 538.048,Z 354.459,A -85,B 0,C 180,E1 -4009.253,E2 -4009.253} C_VEL
LIN {X 0,Y 537.992,Z 354.473,A -85,B 0,C 180,E1 -4012.123,E2 -4012.123} C_VEL
LIN {X 0,Y 538.019,Z 354.462,A -85,B 0,C 180,E1 -4014.918,E2 -4014.918} C_VEL
LIN {X 0,Y 538.031,Z 354.465,A -85,B 0,C 180,E1 -4017.619,E2 -4017.619} C_VEL
LIN {X 0,Y 538.043,Z 354.465,A -85,B 0,C 180,E1 -4020.241,E2 -4020.241} C_VEL
LIN {X 0,Y 538.067,Z 354.458,A -85,B 0,C 180,E1 -4022.797,E2 -4022.797} C_VEL
LIN {X 0,Y 538.072,Z 354.538,A -85,B 0,C 180,E1 -4025.269,E2 -4025.269} C_VEL
LIN {X 0,Y 539.404,Z 361.511,A -85,B 0,C 180,E1 -4026.382,E2 -4026.382} C_VEL
LIN {X 0,Y 539.194,Z 376.356,A -85,B 0,C 180,E1 -4028.595,E2 -4028.595} C_VEL
LIN {X 0,Y 538.784,Z 396.634,A -85,B 0,C 180,E1 -4031.56,E2 -4031.56} C_VEL
LIN {X 0,Y 538.423,Z 416.847,A -85,B 0,C 180,E1 -4034.48,E2 -4034.48} C_VEL
LIN {X 0,Y 538.427,Z 422.435,A -85,B 0,C 180,E1 -4035.251,E2 -4035.251} C_VEL
LIN {X 0,Y 539.704,Z 431.904,A -85,B 0,C 180,E1 -4035.413,E2 -4035.413} C_VEL
LIN {X 0,Y 539.346,Z 530.716,A -85,B 0,C 180,E1 -4036.747,E2 -4036.747} C_VEL
LIN {X 0,Y 539.144,Z 543.248,A -85,B 0,C 180,E1 -4037.053,E2 -4037.053} C_VEL
LIN {X 0,Y 538.939,Z 556.201,A -85,B 0,C 180,E1 -4037.527,E2 -4037.527} C_VEL
LIN {X 0,Y 538.719,Z 568.092,A -85,B 0,C 180,E1 -4038.119,E2 -4038.119} C_VEL
LIN {X 0,Y 538.511,Z 580.134,A -85,B 0,C 180,E1 -4038.902,E2 -4038.902} C_VEL
LIN {X 0,Y 538.262,Z 590.602,A -85,B 0,C 180,E1 -4039.753,E2 -4039.753} C_VEL
LIN {X 0,Y 538.067,Z 599.115,A -85,B 0,C 180,E1 -4040.603,E2 -4040.603} C_VEL
LIN {X 0,Y 537.921,Z 606.962,A -85,B 0,C 180,E1 -4041.548,E2 -4041.548} C_VEL
LIN {X 0,Y 537.754,Z 614.622,A -85,B 0,C 180,E1 -4042.679,E2 -4042.679} C_VEL
LIN {X 0,Y 537.693,Z 621.68,A -85,B 0,C 180,E1 -4043.998,E2 -4043.998} C_VEL
LIN {X 0,Y 537.54,Z 626.373,A -85,B 0,C 180,E1 -4045.125,E2 -4045.125} C_VEL
LIN {X 0,Y 537.591,Z 629.958,A -85,B 0,C 180,E1 -4046.252,E2 -4046.252} C_VEL
LIN {X 0,Y 537.551,Z 631.807,A -85,B 0,C 180,E1 -4047.002,E2 -4047.002} C_VEL
LIN {X 0,Y 537.451,Z 634.182,A -85,B 0,C 180,E1 -4048.501,E2 -4048.501} C_VEL
LIN {X 0,Y 537.442,Z 635,A -85,B 0,C 180,E1 -4050,E2 -4050} C_VEL
LIN {X 0,Y 537.451,Z 634.184,A -85,B 0,C 180,E1 -4051.499,E2 -4051.499} C_VEL
LIN {X 0,Y 537.551,Z 631.81,A -85,B 0,C 180,E1 -4052.998,E2 -4052.998} C_VEL
LIN {X 0,Y 537.603,Z 628.895,A -85,B 0,C 180,E1 -4054.123,E2 -4054.123} C_VEL
LIN {X 0,Y 537.588,Z 624.948,A -85,B 0,C 180,E1 -4055.251,E2 -4055.251} C_VEL
LIN {X 0,Y 537.644,Z 620.125,A -85,B 0,C 180,E1 -4056.326,E2 -4056.326} C_VEL
LIN {X 0,Y 537.79,Z 613.467,A -85,B 0,C 180,E1 -4057.509,E2 -4057.509} C_VEL
LIN {X 0,Y 537.972,Z 605.478,A -85,B 0,C 180,E1 -4058.64,E2 -4058.64} C_VEL
LIN {X 0,Y 538.143,Z 597.335,A -85,B 0,C 180,E1 -4059.585,E2 -4059.585} C_VEL
LIN {X 0,Y 538.383,Z 587.381,A -85,B 0,C 180,E1 -4060.53,E2 -4060.53} C_VEL
LIN {X 0,Y 538.565,Z 577.518,A -85,B 0,C 180,E1 -4061.288,E2 -4061.288} C_VEL
LIN {X 0,Y 538.731,Z 566.412,A -85,B 0,C 180,E1 -4061.973,E2 -4061.973} C_VEL
LIN {X 0,Y 538.966,Z 553.92,A -85,B 0,C 180,E1 -4062.568,E2 -4062.568} C_VEL
LIN {X 0,Y 539.202,Z 540.867,A -85,B 0,C 180,E1 -4063.017,E2 -4063.017} C_VEL
LIN {X 0,Y 539.387,Z 527.861,A -85,B 0,C 180,E1 -4063.3,E2 -4063.3} C_VEL
LIN {X 0,Y 539.548,Z 429.884,A -85,B 0,C 180,E1 -4064.618,E2 -4064.618} C_VEL
LIN {X 0,Y 538.398,Z 422.034,A -85,B 0,C 180,E1 -4064.772,E2 -4064.772} C_VEL
LIN {X 0,Y 538.753,Z 398.999,A -85,B 0,C 180,E1 -4068.09,E2 -4068.09} C_VEL
LIN {X 0,Y 539.158,Z 377.622,A -85,B 0,C 180,E1 -4071.206,E2 -4071.206} C_VEL
LIN {X 0,Y 539.403,Z 361.449,A -85,B 0,C 180,E1 -4073.618,E2 -4073.618} C_VEL
LIN {X 0,Y 538.08,Z 354.461,A -85,B 0,C 180,E1 -4074.757,E2 -4074.757} C_VEL
LIN {X 0,Y 538.061,Z 354.46,A -85,B 0,C 180,E1 -4077.352,E2 -4077.352} C_VEL
LIN {X 0,Y 538.043,Z 354.465,A -85,B 0,C 180,E1 -4079.759,E2 -4079.759} C_VEL
LIN {X 0,Y 538.031,Z 354.465,A -85,B 0,C 180,E1 -4082.381,E2 -4082.381} C_VEL
LIN {X 0,Y 538.019,Z 354.463,A -85,B 0,C 180,E1 -4085.082,E2 -4085.082} C_VEL
LIN {X 0,Y 537.992,Z 354.474,A -85,B 0,C 180,E1 -4087.877,E2 -4087.877} C_VEL
LIN {X 0,Y 538.048,Z 354.458,A -85,B 0,C 180,E1 -4090.775,E2 -4090.775} C_VEL
LIN {X 0,Y 538.02,Z 354.466,A -85,B 0,C 180,E1 -4094.073,E2 -4094.073} C_VEL
LIN {X 0,Y 538.028,Z 354.46,A -85,B 0,C 180,E1 -4097.011,E2 -4097.011} C_VEL
LIN {X 0,Y 538.073,Z 354.457,A -85,B 0,C 180,E1 -4099.248,E2 -4099.248} C_VEL
LIN {X 0,Y 537.989,Z 354.467,A -85,B 0,C 180,E1 -4102.122,E2 -4102.122} C_VEL
LIN {X 0,Y 538.014,Z 354.463,A -85,B 0,C 180,E1 -4104.917,E2 -4104.917} C_VEL
LIN {X 0,Y 538.025,Z 354.469,A -85,B 0,C 180,E1 -4107.618,E2 -4107.618} C_VEL
LIN {X 0,Y 538.036,Z 354.46,A -85,B 0,C 180,E1 -4110.24,E2 -4110.24} C_VEL
LIN {X 0,Y 538.064,Z 354.458,A -85,B 0,C 180,E1 -4112.796,E2 -4112.796} C_VEL
LIN {X 0,Y 538.045,Z 354.46,A -85,B 0,C 180,E1 -4115.292,E2 -4115.292} C_VEL
LIN {X 0,Y 538.023,Z 354.462,A -85,B 0,C 180,E1 -4118.037,E2 -4118.037} C_VEL
LIN {X 0,Y 538.033,Z 354.464,A -85,B 0,C 180,E1 -4120.94,E2 -4120.94} C_VEL
LIN {X 0,Y 538.021,Z 354.469,A -85,B 0,C 180,E1 -4123.299,E2 -4123.299} C_VEL
LIN {X 0,Y 538.055,Z 354.46,A -85,B 0,C 180,E1 -4125.631,E2 -4125.631} C_VEL
LIN {X 0,Y 538.088,Z 354.457,A -85,B 0,C 180,E1 -4128.702,E2 -4128.702} C_VEL
LIN {X 0,Y 538.084,Z 354.455,A -85,B 0,C 180,E1 -4131.74,E2 -4131.74} C_VEL
LIN {X 0,Y 538.158,Z 354.449,A -85,B 0,C 180,E1 -4134.755,E2 -4134.755} C_VEL
LIN {X 0,Y 538.159,Z 354.444,A -85,B 0,C 180,E1 -4137.755,E2 -4137.755} C_VEL
LIN {X 0,Y 538.18,Z 354.449,A -85,B 0,C 180,E1 -4140.748,E2 -4140.748} C_VEL
LIN {X 0,Y 538.137,Z 354.452,A -85,B 0,C 180,E1 -4142.995,E2 -4142.995} C_VEL
LIN {X 0,Y 538.116,Z 354.451,A -85,B 0,C 180,E1 -4145.998,E2 -4145.998} C_VEL
LIN {X 0,Y 538.069,Z 354.46,A -85,B 0,C 180,E1 -4149.018,E2 -4149.018} C_VEL
LIN {X 0,Y 538.076,Z 354.456,A -85,B 0,C 180,E1 -4152.063,E2 -4152.063} C_VEL
LIN {X 0,Y 538.037,Z 354.461,A -85,B 0,C 180,E1 -4155.144,E2 -4155.144} C_VEL
LIN {X 0,Y 538.027,Z 354.466,A -85,B 0,C 180,E1 -4158.271,E2 -4158.271} C_VEL
LIN {X 0,Y 538.035,Z 354.465,A -85,B 0,C 180,E1 -4160.652,E2 -4160.652} C_VEL
LIN {X 0,Y 538.017,Z 354.465,A -85,B 0,C 180,E1 -4163.888,E2 -4163.888} C_VEL
LIN {X 0,Y 538.043,Z 354.462,A -85,B 0,C 180,E1 -4166.367,E2 -4166.367} C_VEL
LIN {X 0,Y 538.025,Z 354.462,A -85,B 0,C 180,E1 -4168.935,E2 -4168.935} C_VEL
LIN {X 0,Y 538.022,Z 354.465,A -85,B 0,C 180,E1 -4171.891,E2 -4171.891} C_VEL
LIN {X 0,Y 538.026,Z 354.464,A -85,B 0,C 180,E1 -4174.622,E2 -4174.622} C_VEL
LIN {X 0,Y 538.004,Z 354.464,A -85,B 0,C 180,E1 -4177.172,E2 -4177.172} C_VEL
LIN {X 0,Y 538.045,Z 354.46,A -85,B 0,C 180,E1 -4180.281,E2 -4180.281} C_VEL
LIN {X 0,Y 537.394,Z 354.543,A -85,B 0,C 180,E1 -4180.906,E2 -4180.906} C_VEL
LIN {X 0,Y 534.533,Z 354.904,A -85,B 0,C 180,E1 -4181.921,E2 -4181.921} C_VEL
LIN {X 0,Y 532.1,Z 355.206,A -85,B 0,C 180,E1 -4182.738,E2 -4182.738} C_VEL
LIN {X 0,Y 531.049,Z 355.334,A -85,B 0,C 180,E1 -4183.369,E2 -4183.369} C_VEL
LIN {X 0,Y 530.96,Z 355.344,A -85,B 0,C 180,E1 -4183.582,E2 -4183.582} C_VEL
LIN {X 0,Y 530.96,Z 355.345,A -85,B 0,C 180,E1 -4186.506,E2 -4186.506} C_VEL
LIN {X 0,Y 531.026,Z 355.34,A -85,B 0,C 180,E1 -4189.572,E2 -4189.572} C_VEL
LIN {X 0,Y 530.97,Z 355.342,A -85,B 0,C 180,E1 -4192.578,E2 -4192.578} C_VEL
LIN {X 0,Y 531.003,Z 355.34,A -85,B 0,C 180,E1 -4195.312,E2 -4195.312} C_VEL
LIN {X 0,Y 530.973,Z 355.346,A -85,B 0,C 180,E1 -4198.033,E2 -4198.033} C_VEL
LIN {X 0,Y 530.999,Z 355.34,A -85,B 0,C 180,E1 -4200.874,E2 -4200.874} C_VEL
LIN {X 0,Y 531.034,Z 355.374,A -85,B 0,C 180,E1 -4201.978,E2 -4201.978} C_VEL
LIN {X 0,Y 531.518,Z 360.611,A -85,B 0,C 180,E1 -4203.073,E2 -4203.073} C_VEL
LIN {X 0,Y 531.175,Z 375.537,A -85,B 0,C 180,E1 -4206.111,E2 -4206.111} C_VEL
LIN {X 0,Y 532.85,Z 385.174,A -85,B 0,C 180,E1 -4206.294,E2 -4206.294} C_VEL
LIN {X 0,Y 532.4,Z 482.436,A -85,B 0,C 180,E1 -4207.632,E2 -4207.632} C_VEL
LIN {X 0,Y 532.215,Z 495.784,A -85,B 0,C 180,E1 -4207.979,E2 -4207.979} C_VEL
LIN {X 0,Y 532.028,Z 507.922,A -85,B 0,C 180,E1 -4208.445,E2 -4208.445} C_VEL
LIN {X 0,Y 531.81,Z 518.652,A -85,B 0,C 180,E1 -4208.995,E2 -4208.995} C_VEL
LIN {X 0,Y 531.594,Z 529.643,A -85,B 0,C 180,E1 -4209.714,E2 -4209.714} C_VEL
LIN {X 0,Y 531.3,Z 540.335,A -85,B 0,C 180,E1 -4210.589,E2 -4210.589} C_VEL
LIN {X 0,Y 531.082,Z 549.22,A -85,B 0,C 180,E1 -4211.483,E2 -4211.483} C_VEL
LIN {X 0,Y 530.888,Z 557.593,A -85,B 0,C 180,E1 -4212.507,E2 -4212.507} C_VEL
LIN {X 0,Y 530.729,Z 565.166,A -85,B 0,C 180,E1 -4213.657,E2 -4213.657} C_VEL
LIN {X 0,Y 530.594,Z 572.143,A -85,B 0,C 180,E1 -4214.995,E2 -4214.995} C_VEL
LIN {X 0,Y 530.503,Z 577.006,A -85,B 0,C 180,E1 -4216.205,E2 -4216.205} C_VEL
LIN {X 0,Y 530.473,Z 579.464,A -85,B 0,C 180,E1 -4216.984,E2 -4216.984} C_VEL
LIN {X 0,Y 530.409,Z 581.46,A -85,B 0,C 180,E1 -4217.761,E2 -4217.761} C_VEL
LIN {X 0,Y 530.451,Z 583.221,A -85,B 0,C 180,E1 -4218.65,E2 -4218.65} C_VEL
LIN {X 0,Y 530.39,Z 584.84,A -85,B 0,C 180,E1 -4220.081,E2 -4220.081} C_VEL
LIN {X 0,Y 530.418,Z 585.064,A -85,B 0,C 180,E1 -4221.62,E2 -4221.62} C_VEL
LIN {X 0,Y 530.428,Z 584.553,A -85,B 0,C 180,E1 -4222.386,E2 -4222.386} C_VEL
LIN {X 0,Y 530.478,Z 583.055,A -85,B 0,C 180,E1 -4223.535,E2 -4223.535} C_VEL
LIN {X 0,Y 530.434,Z 579.59,A -85,B 0,C 180,E1 -4225.06,E2 -4225.06} C_VEL
LIN {X 0,Y 530.534,Z 575.829,A -85,B 0,C 180,E1 -4226.202,E2 -4226.202} C_VEL
LIN {X 0,Y 530.593,Z 570.973,A -85,B 0,C 180,E1 -4227.343,E2 -4227.343} C_VEL
LIN {X 0,Y 530.686,Z 564.879,A -85,B 0,C 180,E1 -4228.482,E2 -4228.482} C_VEL
LIN {X 0,Y 530.897,Z 557.296,A -85,B 0,C 180,E1 -4229.621,E2 -4229.621} C_VEL
LIN {X 0,Y 531.112,Z 547.815,A -85,B 0,C 180,E1 -4230.758,E2 -4230.758} C_VEL
LIN {X 0,Y 531.332,Z 538.061,A -85,B 0,C 180,E1 -4231.705,E2 -4231.705} C_VEL
LIN {X 0,Y 531.563,Z 527.1,A -85,B 0,C 180,E1 -4232.557,E2 -4232.557} C_VEL
LIN {X 0,Y 531.815,Z 516.39,A -85,B 0,C 180,E1 -4233.22,E2 -4233.22} C_VEL
LIN {X 0,Y 532.03,Z 504.607,A -85,B 0,C 180,E1 -4233.787,E2 -4233.787} C_VEL
LIN {X 0,Y 532.259,Z 491.757,A -85,B 0,C 180,E1 -4234.236,E2 -4234.236} C_VEL
LIN {X 0,Y 532.415,Z 479.015,A -85,B 0,C 180,E1 -4234.519,E2 -4234.519} C_VEL
LIN {X 0,Y 532.737,Z 383.571,A -85,B 0,C 180,E1 -4235.821,E2 -4235.821} C_VEL
LIN {X 0,Y 531.281,Z 375.504,A -85,B 0,C 180,E1 -4235.979,E2 -4235.979} C_VEL
LIN {X 0,Y 531.502,Z 360.001,A -85,B 0,C 180,E1 -4239.13,E2 -4239.13} C_VEL
LIN {X 0,Y 531.01,Z 355.344,A -85,B 0,C 180,E1 -4240.148,E2 -4240.148} C_VEL
LIN {X 0,Y 531.047,Z 355.339,A -85,B 0,C 180,E1 -4242.225,E2 -4242.225} C_VEL
LIN {X 0,Y 531.001,Z 355.336,A -85,B 0,C 180,E1 -4245.349,E2 -4245.349} C_VEL
LIN {X 0,Y 530.993,Z 355.344,A -85,B 0,C 180,E1 -4248.521,E2 -4248.521} C_VEL
LIN {X 0,Y 531.003,Z 355.337,A -85,B 0,C 180,E1 -4250.937,E2 -4250.937} C_VEL
LIN {X 0,Y 530.984,Z 355.347,A -85,B 0,C 180,E1 -4254.224,E2 -4254.224} C_VEL
LIN {X 0,Y 531.009,Z 355.337,A -85,B 0,C 180,E1 -4256.743,E2 -4256.743} C_VEL
LIN {X 0,Y 531.003,Z 355.337,A -85,B 0,C 180,E1 -4259.321,E2 -4259.321} C_VEL
LIN {X 0,Y 530.972,Z 355.348,A -85,B 0,C 180,E1 -4262.1,E2 -4262.1} C_VEL
LIN {X 0,Y 530.99,Z 355.339,A -85,B 0,C 180,E1 -4264.853,E2 -4264.853} C_VEL
LIN {X 0,Y 530.967,Z 355.344,A -85,B 0,C 180,E1 -4267.507,E2 -4267.507} C_VEL
LIN {X 0,Y 530.983,Z 355.342,A -85,B 0,C 180,E1 -4270.432,E2 -4270.432} C_VEL
LIN {X 0,Y 530.963,Z 355.346,A -85,B 0,C 180,E1 -4273.494,E2 -4273.494} C_VEL
LIN {X 0,Y 530.964,Z 355.343,A -85,B 0,C 180,E1 -4276.505,E2 -4276.505} C_VEL
LIN {X 0,Y 531.023,Z 355.34,A -85,B 0,C 180,E1 -4279.57,E2 -4279.57} C_VEL
LIN {X 0,Y 530.964,Z 355.342,A -85,B 0,C 180,E1 -4282.576,E2 -4282.576} C_VEL
LIN {X 0,Y 530.991,Z 355.343,A -85,B 0,C 180,E1 -4285.31,E2 -4285.31} C_VEL
LIN {X 0,Y 530.977,Z 355.344,A -85,B 0,C 180,E1 -4288.032,E2 -4288.032} C_VEL
LIN {X 0,Y 530.983,Z 355.341,A -85,B 0,C 180,E1 -4290.873,E2 -4290.873} C_VEL
LIN {X 0,Y 531.005,Z 355.342,A -85,B 0,C 180,E1 -4293.256,E2 -4293.256} C_VEL
LIN {X 0,Y 531.001,Z 355.34,A -85,B 0,C 180,E1 -4295.954,E2 -4295.954} C_VEL
LIN {X 0,Y 530.998,Z 355.342,A -85,B 0,C 180,E1 -4299.062,E2 -4299.062} C_VEL
LIN {X 0,Y 531.008,Z 355.337,A -85,B 0,C 180,E1 -4302.277,E2 -4302.277} C_VEL
LIN {X 0,Y 531.032,Z 355.34,A -85,B 0,C 180,E1 -4305.436,E2 -4305.436} C_VEL
LIN {X 0,Y 531.038,Z 355.334,A -85,B 0,C 180,E1 -4308.549,E2 -4308.549} C_VEL
LIN {X 0,Y 531.053,Z 355.334,A -85,B 0,C 180,E1 -4311.629,E2 -4311.629} C_VEL
LIN {X 0,Y 531.117,Z 355.327,A -85,B 0,C 180,E1 -4314.685,E2 -4314.685} C_VEL
LIN {X 0,Y 531.132,Z 355.323,A -85,B 0,C 180,E1 -4317.725,E2 -4317.725} C_VEL
LIN {X 0,Y 531.149,Z 355.325,A -85,B 0,C 180,E1 -4320.758,E2 -4320.758} C_VEL
LIN {X 0,Y 531.103,Z 355.331,A -85,B 0,C 180,E1 -4323.034,E2 -4323.034} C_VEL
LIN {X 0,Y 531.076,Z 355.329,A -85,B 0,C 180,E1 -4326.077,E2 -4326.077} C_VEL
LIN {X 0,Y 531.029,Z 355.339,A -85,B 0,C 180,E1 -4329.138,E2 -4329.138} C_VEL
LIN {X 0,Y 531.032,Z 355.336,A -85,B 0,C 180,E1 -4332.225,E2 -4332.225} C_VEL
LIN {X 0,Y 530.988,Z 355.341,A -85,B 0,C 180,E1 -4335.35,E2 -4335.35} C_VEL
LIN {X 0,Y 531.007,Z 355.337,A -85,B 0,C 180,E1 -4337.723,E2 -4337.723} C_VEL
LIN {X 0,Y 530.996,Z 355.343,A -85,B 0,C 180,E1 -4340.938,E2 -4340.938} C_VEL
LIN {X 0,Y 530.999,Z 355.34,A -85,B 0,C 180,E1 -4344.045,E2 -4344.045} C_VEL
LIN {X 0,Y 531.004,Z 355.342,A -85,B 0,C 180,E1 -4346.744,E2 -4346.744} C_VEL
LIN {X 0,Y 530.975,Z 355.341,A -85,B 0,C 180,E1 -4349.323,E2 -4349.323} C_VEL
LIN {X 0,Y 530.973,Z 355.345,A -85,B 0,C 180,E1 -4352.104,E2 -4352.104} C_VEL
LIN {X 0,Y 530.984,Z 355.342,A -85,B 0,C 180,E1 -4354.855,E2 -4354.855} C_VEL
LIN {X 0,Y 530.961,Z 355.342,A -85,B 0,C 180,E1 -4357.508,E2 -4357.508} C_VEL
LIN {X 0,Y 531.021,Z 355.34,A -85,B 0,C 180,E1 -4360.429,E2 -4360.429} C_VEL
LIN {X 0,Y 530.961,Z 355.343,A -85,B 0,C 180,E1 -4363.495,E2 -4363.495} C_VEL
LIN {X 0,Y 530.96,Z 355.346,A -85,B 0,C 180,E1 -4366.506,E2 -4366.506} C_VEL
LIN {X 0,Y 530.986,Z 355.339,A -85,B 0,C 180,E1 -4368.976,E2 -4368.976} C_VEL
LIN {X 0,Y 530.957,Z 355.344,A -85,B 0,C 180,E1 -4371.53,E2 -4371.53} C_VEL
LIN {X 0,Y 530.981,Z 355.343,A -85,B 0,C 180,E1 -4374.383,E2 -4374.383} C_VEL
LIN {X 0,Y 530.972,Z 355.34,A -85,B 0,C 180,E1 -4377.135,E2 -4377.135} C_VEL
LIN {X 0,Y 530.987,Z 355.346,A -85,B 0,C 180,E1 -4379.805,E2 -4379.805} C_VEL
LIN {X 0,Y 531.016,Z 355.338,A -85,B 0,C 180,E1 -4382.467,E2 -4382.467} C_VEL
LIN {X 0,Y 531.047,Z 355.452,A -85,B 0,C 180,E1 -4385.102,E2 -4385.102} C_VEL
LIN {X 0,Y 532.545,Z 363.936,A -85,B 0,C 180,E1 -4386.472,E2 -4386.472} C_VEL
LIN {X 0,Y 532.068,Z 382.742,A -85,B 0,C 180,E1 -4389.302,E2 -4389.302} C_VEL
LIN {X 0,Y 531.707,Z 401.797,A -85,B 0,C 180,E1 -4392.117,E2 -4392.117} C_VEL
LIN {X 0,Y 531.376,Z 421.817,A -85,B 0,C 180,E1 -4395.043,E2 -4395.043} C_VEL
LIN {X 0,Y 532.821,Z 432.385,A -85,B 0,C 180,E1 -4395.231,E2 -4395.231} C_VEL
LIN {X 0,Y 532.43,Z 530.366,A -85,B 0,C 180,E1 -4396.572,E2 -4396.572} C_VEL
LIN {X 0,Y 532.192,Z 543.668,A -85,B 0,C 180,E1 -4396.906,E2 -4396.906} C_VEL
LIN {X 0,Y 531.983,Z 555.86,A -85,B 0,C 180,E1 -4397.361,E2 -4397.361} C_VEL
LIN {X 0,Y 531.726,Z 568.135,A -85,B 0,C 180,E1 -4397.983,E2 -4397.983} C_VEL
LIN {X 0,Y 531.502,Z 579.796,A -85,B 0,C 180,E1 -4398.753,E2 -4398.753} C_VEL
LIN {X 0,Y 531.22,Z 590.269,A -85,B 0,C 180,E1 -4399.615,E2 -4399.615} C_VEL
LIN {X 0,Y 531.033,Z 598.836,A -85,B 0,C 180,E1 -4400.478,E2 -4400.478} C_VEL
LIN {X 0,Y 530.886,Z 606.744,A -85,B 0,C 180,E1 -4401.435,E2 -4401.435} C_VEL
LIN {X 0,Y 530.681,Z 614.466,A -85,B 0,C 180,E1 -4402.581,E2 -4402.581} C_VEL
LIN {X 0,Y 530.604,Z 621.589,A -85,B 0,C 180,E1 -4403.918,E2 -4403.918} C_VEL
LIN {X 0,Y 530.459,Z 626.325,A -85,B 0,C 180,E1 -4405.06,E2 -4405.06} C_VEL
LIN {X 0,Y 530.516,Z 629.947,A -85,B 0,C 180,E1 -4406.202,E2 -4406.202} C_VEL
LIN {X 0,Y 530.457,Z 631.804,A -85,B 0,C 180,E1 -4406.962,E2 -4406.962} C_VEL
LIN {X 0,Y 530.41,Z 633.192,A -85,B 0,C 180,E1 -4407.722,E2 -4407.722} C_VEL
LIN {X 0,Y 530.344,Z 634.785,A -85,B 0,C 180,E1 -4409.241,E2 -4409.241} C_VEL
LIN {X 0,Y 530.342,Z 635,A -85,B 0,C 180,E1 -4410,E2 -4410} C_VEL
LIN {X 0,Y 530.361,Z 634.183,A -85,B 0,C 180,E1 -4411.519,E2 -4411.519} C_VEL
LIN {X 0,Y 530.41,Z 633.195,A -85,B 0,C 180,E1 -4412.278,E2 -4412.278} C_VEL
LIN {X 0,Y 530.457,Z 631.807,A -85,B 0,C 180,E1 -4413.038,E2 -4413.038} C_VEL
LIN {X 0,Y 530.522,Z 628.876,A -85,B 0,C 180,E1 -4414.178,E2 -4414.178} C_VEL
LIN {X 0,Y 530.525,Z 624.887,A -85,B 0,C 180,E1 -4415.321,E2 -4415.321} C_VEL
LIN {X 0,Y 530.595,Z 619.162,A -85,B 0,C 180,E1 -4416.579,E2 -4416.579} C_VEL
LIN {X 0,Y 530.733,Z 612.056,A -85,B 0,C 180,E1 -4417.801,E2 -4417.801} C_VEL
LIN {X 0,Y 530.93,Z 603.746,A -85,B 0,C 180,E1 -4418.948,E2 -4418.948} C_VEL
LIN {X 0,Y 531.122,Z 595.231,A -85,B 0,C 180,E1 -4419.905,E2 -4419.905} C_VEL
LIN {X 0,Y 531.38,Z 584.713,A -85,B 0,C 180,E1 -4420.863,E2 -4420.863} C_VEL
LIN {X 0,Y 531.66,Z 572.745,A -85,B 0,C 180,E1 -4421.735,E2 -4421.735} C_VEL
LIN {X 0,Y 531.927,Z 560.985,A -85,B 0,C 180,E1 -4422.398,E2 -4422.398} C_VEL
LIN {X 0,Y 532.135,Z 548.615,A -85,B 0,C 180,E1 -4422.926,E2 -4422.926} C_VEL
LIN {X 0,Y 532.339,Z 535.928,A -85,B 0,C 180,E1 -4423.309,E2 -4423.309} C_VEL
LIN {X 0,Y 532.484,Z 522.688,A -85,B 0,C 180,E1 -4423.548,E2 -4423.548} C_VEL
LIN {X 0,Y 532.718,Z 430.886,A -85,B 0,C 180,E1 -4424.792,E2 -4424.792} C_VEL
LIN {X 0,Y 531.34,Z 421.73,A -85,B 0,C 180,E1 -4424.966,E2 -4424.966} C_VEL
LIN {X 0,Y 531.743,Z 400.117,A -85,B 0,C 180,E1 -4428.125,E2 -4428.125} C_VEL
LIN {X 0,Y 532.137,Z 380.051,A -85,B 0,C 180,E1 -4431.093,E2 -4431.093} C_VEL
LIN {X 0,Y 532.549,Z 363.865,A -85,B 0,C 180,E1 -4433.528,E2 -4433.528} C_VEL
LIN {X 0,Y 531.053,Z 355.335,A -85,B 0,C 180,E1 -4434.924,E2 -4434.924} C_VEL
LIN {X 0,Y 531.017,Z 355.339,A -85,B 0,C 180,E1 -4437.595,E2 -4437.595} C_VEL
LIN {X 0,Y 530.982,Z 355.339,A -85,B 0,C 180,E1 -4440.646,E2 -4440.646} C_VEL
LIN {X 0,Y 530.99,Z 355.344,A -85,B 0,C 180,E1 -4443.772,E2 -4443.772} C_VEL
LIN {X 0,Y 530.967,Z 355.343,A -85,B 0,C 180,E1 -4446.557,E2 -4446.557} C_VEL
LIN {X 0,Y 530.981,Z 355.347,A -85,B 0,C 180,E1 -4449.854,E2 -4449.854} C_VEL
LIN {X 0,Y 530.977,Z 355.34,A -85,B 0,C 180,E1 -4452.456,E2 -4452.456} C_VEL
LIN {X 0,Y 530.983,Z 355.345,A -85,B 0,C 180,E1 -4455.62,E2 -4455.62} C_VEL
LIN {X 0,Y 531.002,Z 355.335,A -85,B 0,C 180,E1 -4458.565,E2 -4458.565} C_VEL
LIN {X 0,Y 530.963,Z 355.345,A -85,B 0,C 180,E1 -4461.345,E2 -4461.345} C_VEL
LIN {X 0,Y 530.976,Z 355.339,A -85,B 0,C 180,E1 -4464.382,E2 -4464.382} C_VEL
LIN {X 0,Y 530.968,Z 355.344,A -85,B 0,C 180,E1 -4467.133,E2 -4467.133} C_VEL
LIN {X 0,Y 530.979,Z 355.343,A -85,B 0,C 180,E1 -4469.804,E2 -4469.804} C_VEL
LIN {X 0,Y 531.01,Z 355.335,A -85,B 0,C 180,E1 -4472.466,E2 -4472.466} C_VEL
LIN {X 0,Y 531.002,Z 355.334,A -85,B 0,C 180,E1 -4474.942,E2 -4474.942} C_VEL
LIN {X 0,Y 530.983,Z 355.34,A -85,B 0,C 180,E1 -4477.893,E2 -4477.893} C_VEL
LIN {X 0,Y 530.989,Z 355.338,A -85,B 0,C 180,E1 -4480.677,E2 -4480.677} C_VEL
LIN {X 0,Y 530.986,Z 355.345,A -85,B 0,C 180,E1 -4483.071,E2 -4483.071} C_VEL
LIN {X 0,Y 531.01,Z 355.34,A -85,B 0,C 180,E1 -4485.436,E2 -4485.436} C_VEL
LIN {X 0,Y 531.043,Z 355.333,A -85,B 0,C 180,E1 -4488.55,E2 -4488.55} C_VEL
LIN {X 0,Y 531.053,Z 355.332,A -85,B 0,C 180,E1 -4491.63,E2 -4491.63} C_VEL
LIN {X 0,Y 531.117,Z 355.324,A -85,B 0,C 180,E1 -4494.685,E2 -4494.685} C_VEL
LIN {X 0,Y 531.131,Z 355.319,A -85,B 0,C 180,E1 -4497.725,E2 -4497.725} C_VEL
LIN {X 0,Y 531.149,Z 355.325,A -85,B 0,C 180,E1 -4500.758,E2 -4500.758} C_VEL
LIN {X 0,Y 531.103,Z 355.327,A -85,B 0,C 180,E1 -4503.034,E2 -4503.034} C_VEL
LIN {X 0,Y 531.076,Z 355.328,A -85,B 0,C 180,E1 -4506.077,E2 -4506.077} C_VEL
LIN {X 0,Y 531.028,Z 355.335,A -85,B 0,C 180,E1 -4509.138,E2 -4509.138} C_VEL
LIN {X 0,Y 531.033,Z 355.335,A -85,B 0,C 180,E1 -4512.225,E2 -4512.225} C_VEL
LIN {X 0,Y 530.988,Z 355.338,A -85,B 0,C 180,E1 -4515.35,E2 -4515.35} C_VEL
LIN {X 0,Y 531.008,Z 355.335,A -85,B 0,C 180,E1 -4517.723,E2 -4517.723} C_VEL
LIN {X 0,Y 530.994,Z 355.338,A -85,B 0,C 180,E1 -4520.938,E2 -4520.938} C_VEL
LIN {X 0,Y 530.973,Z 355.347,A -85,B 0,C 180,E1 -4524.225,E2 -4524.225} C_VEL
LIN {X 0,Y 531.005,Z 355.335,A -85,B 0,C 180,E1 -4526.744,E2 -4526.744} C_VEL
LIN {X 0,Y 530.976,Z 355.34,A -85,B 0,C 180,E1 -4529.323,E2 -4529.323} C_VEL
LIN {X 0,Y 530.975,Z 355.346,A -85,B 0,C 180,E1 -4532.104,E2 -4532.104} C_VEL
LIN {X 0,Y 530.983,Z 355.34,A -85,B 0,C 180,E1 -4534.855,E2 -4534.855} C_VEL
LIN {X 0,Y 530.963,Z 355.343,A -85,B 0,C 180,E1 -4537.508,E2 -4537.508} C_VEL
LIN {X 0,Y 531.023,Z 355.338,A -85,B 0,C 180,E1 -4540.43,E2 -4540.43} C_VEL
LIN {X 0,Y 530.96,Z 355.344,A -85,B 0,C 180,E1 -4543.582,E2 -4543.582} C_VEL
LIN {X 0,Y 530.288,Z 355.433,A -85,B 0,C 180,E1 -4544.216,E2 -4544.216} C_VEL
LIN {X 0,Y 527.438,Z 355.783,A -85,B 0,C 180,E1 -4545.245,E2 -4545.245} C_VEL
LIN {X 0,Y 525.033,Z 356.087,A -85,B 0,C 180,E1 -4546.073,E2 -4546.073} C_VEL
LIN {X 0,Y 524.001,Z 356.211,A -85,B 0,C 180,E1 -4546.713,E2 -4546.713} C_VEL
LIN {X 0,Y 523.917,Z 356.22,A -85,B 0,C 180,E1 -4546.929,E2 -4546.929} C_VEL
LIN {X 0,Y 523.978,Z 356.22,A -85,B 0,C 180,E1 -4549.924,E2 -4549.924} C_VEL
LIN {X 0,Y 523.912,Z 356.221,A -85,B 0,C 180,E1 -4552.869,E2 -4552.869} C_VEL
LIN {X 0,Y 523.946,Z 356.223,A -85,B 0,C 180,E1 -4555.712,E2 -4555.712} C_VEL
LIN {X 0,Y 523.926,Z 356.221,A -85,B 0,C 180,E1 -4558.457,E2 -4558.457} C_VEL
LIN {X 0,Y 523.962,Z 356.222,A -85,B 0,C 180,E1 -4561.565,E2 -4561.565} C_VEL
LIN {X 0,Y 523.986,Z 356.24,A -85,B 0,C 180,E1 -4561.839,E2 -4561.839} C_VEL
LIN {X 0,Y 524.542,Z 361.228,A -85,B 0,C 180,E1 -4562.901,E2 -4562.901} C_VEL
LIN {X 0,Y 524.197,Z 375.836,A -85,B 0,C 180,E1 -4565.898,E2 -4565.898} C_VEL
LIN {X 0,Y 525.999,Z 385.682,A -85,B 0,C 180,E1 -4566.1,E2 -4566.1} C_VEL
LIN {X 0,Y 525.531,Z 482.098,A -85,B 0,C 180,E1 -4567.439,E2 -4567.439} C_VEL
LIN {X 0,Y 525.348,Z 494.921,A -85,B 0,C 180,E1 -4567.767,E2 -4567.767} C_VEL
LIN {X 0,Y 525.135,Z 507.653,A -85,B 0,C 180,E1 -4568.251,E2 -4568.251} C_VEL
LIN {X 0,Y 524.863,Z 520.215,A -85,B 0,C 180,E1 -4568.909,E2 -4568.909} C_VEL
LIN {X 0,Y 524.572,Z 531.699,A -85,B 0,C 180,E1 -4569.692,E2 -4569.692} C_VEL
LIN {X 0,Y 524.269,Z 542.558,A -85,B 0,C 180,E1 -4570.624,E2 -4570.624} C_VEL
LIN {X 0,Y 524.012,Z 551.926,A -85,B 0,C 180,E1 -4571.629,E2 -4571.629} C_VEL
LIN {X 0,Y 523.763,Z 560.981,A -85,B 0,C 180,E1 -4572.831,E2 -4572.831} C_VEL
LIN {X 0,Y 523.588,Z 568.146,A -85,B 0,C 180,E1 -4574.028,E2 -4574.028} C_VEL
LIN {X 0,Y 523.514,Z 573.813,A -85,B 0,C 180,E1 -4575.223,E2 -4575.223} C_VEL
LIN {X 0,Y 523.418,Z 578.221,A -85,B 0,C 180,E1 -4576.41,E2 -4576.41} C_VEL
LIN {X 0,Y 523.356,Z 581.511,A -85,B 0,C 180,E1 -4577.593,E2 -4577.593} C_VEL
LIN {X 0,Y 523.366,Z 583.536,A -85,B 0,C 180,E1 -4578.605,E2 -4578.605} C_VEL
LIN {X 0,Y 523.31,Z 585.099,A -85,B 0,C 180,E1 -4579.946,E2 -4579.946} C_VEL
LIN {X 0,Y 523.339,Z 585.423,A -85,B 0,C 180,E1 -4581.505,E2 -4581.505} C_VEL
LIN {X 0,Y 523.357,Z 585.002,A -85,B 0,C 180,E1 -4582.283,E2 -4582.283} C_VEL
LIN {X 0,Y 523.388,Z 583.418,A -85,B 0,C 180,E1 -4583.552,E2 -4583.552} C_VEL
LIN {X 0,Y 523.355,Z 580.252,A -85,B 0,C 180,E1 -4584.993,E2 -4584.993} C_VEL
LIN {X 0,Y 523.458,Z 576.602,A -85,B 0,C 180,E1 -4586.151,E2 -4586.151} C_VEL
LIN {X 0,Y 523.539,Z 571.863,A -85,B 0,C 180,E1 -4587.307,E2 -4587.307} C_VEL
LIN {X 0,Y 523.661,Z 564.797,A -85,B 0,C 180,E1 -4588.654,E2 -4588.654} C_VEL
LIN {X 0,Y 523.868,Z 557.085,A -85,B 0,C 180,E1 -4589.808,E2 -4589.808} C_VEL
LIN {X 0,Y 524.13,Z 547.491,A -85,B 0,C 180,E1 -4590.96,E2 -4590.96} C_VEL
LIN {X 0,Y 524.368,Z 537.581,A -85,B 0,C 180,E1 -4591.92,E2 -4591.92} C_VEL
LIN {X 0,Y 524.63,Z 526.385,A -85,B 0,C 180,E1 -4592.783,E2 -4592.783} C_VEL
LIN {X 0,Y 524.949,Z 515.409,A -85,B 0,C 180,E1 -4593.454,E2 -4593.454} C_VEL
LIN {X 0,Y 525.14,Z 503.252,A -85,B 0,C 180,E1 -4594.029,E2 -4594.029} C_VEL
LIN {X 0,Y 525.355,Z 490.31,A -85,B 0,C 180,E1 -4594.46,E2 -4594.46} C_VEL
LIN {X 0,Y 525.557,Z 477.85,A -85,B 0,C 180,E1 -4594.722,E2 -4594.722} C_VEL
LIN {X 0,Y 525.953,Z 384.717,A -85,B 0,C 180,E1 -4596.004,E2 -4596.004} C_VEL
LIN {X 0,Y 524.294,Z 375.853,A -85,B 0,C 180,E1 -4596.18,E2 -4596.18} C_VEL
LIN {X 0,Y 524.515,Z 360.862,A -85,B 0,C 180,E1 -4599.252,E2 -4599.252} C_VEL
LIN {X 0,Y 523.995,Z 356.218,A -85,B 0,C 180,E1 -4600.285,E2 -4600.285} C_VEL
LIN {X 0,Y 523.983,Z 356.22,A -85,B 0,C 180,E1 -4602.392,E2 -4602.392} C_VEL
LIN {X 0,Y 523.946,Z 356.215,A -85,B 0,C 180,E1 -4605.561,E2 -4605.561} C_VEL
LIN {X 0,Y 523.969,Z 356.216,A -85,B 0,C 180,E1 -4607.968,E2 -4607.968} C_VEL
LIN {X 0,Y 523.976,Z 356.219,A -85,B 0,C 180,E1 -4610.409,E2 -4610.409} C_VEL
LIN {X 0,Y 523.921,Z 356.22,A -85,B 0,C 180,E1 -4612.893,E2 -4612.893} C_VEL
LIN {X 0,Y 523.957,Z 356.215,A -85,B 0,C 180,E1 -4615.418,E2 -4615.418} C_VEL
LIN {X 0,Y 523.973,Z 356.218,A -85,B 0,C 180,E1 -4617.998,E2 -4617.998} C_VEL
LIN {X 0,Y 523.952,Z 356.216,A -85,B 0,C 180,E1 -4620.855,E2 -4620.855} C_VEL
LIN {X 0,Y 523.963,Z 356.218,A -85,B 0,C 180,E1 -4623.734,E2 -4623.734} C_VEL
LIN {X 0,Y 523.924,Z 356.222,A -85,B 0,C 180,E1 -4626.403,E2 -4626.403} C_VEL
LIN {X 0,Y 523.922,Z 356.219,A -85,B 0,C 180,E1 -4629.084,E2 -4629.084} C_VEL
LIN {X 0,Y 523.951,Z 356.221,A -85,B 0,C 180,E1 -4632.118,E2 -4632.118} C_VEL
LIN {X 0,Y 523.954,Z 356.217,A -85,B 0,C 180,E1 -4635.308,E2 -4635.308} C_VEL
LIN {X 0,Y 523.969,Z 356.214,A -85,B 0,C 180,E1 -4638.687,E2 -4638.687} C_VEL
LIN {X 0,Y 523.921,Z 356.221,A -85,B 0,C 180,E1 -4641.078,E2 -4641.078} C_VEL
LIN {X 0,Y 523.92,Z 356.227,A -85,B 0,C 180,E1 -4643.826,E2 -4643.826} C_VEL
LIN {X 0,Y 523.937,Z 356.218,A -85,B 0,C 180,E1 -4646.635,E2 -4646.635} C_VEL
LIN {X 0,Y 523.951,Z 356.221,A -85,B 0,C 180,E1 -4649.355,E2 -4649.355} C_VEL
LIN {X 0,Y 523.974,Z 356.214,A -85,B 0,C 180,E1 -4652.28,E2 -4652.28} C_VEL
LIN {X 0,Y 523.949,Z 356.216,A -85,B 0,C 180,E1 -4654.581,E2 -4654.581} C_VEL
LIN {X 0,Y 523.937,Z 356.222,A -85,B 0,C 180,E1 -4657.107,E2 -4657.107} C_VEL
LIN {X 0,Y 523.971,Z 356.216,A -85,B 0,C 180,E1 -4659.865,E2 -4659.865} C_VEL
LIN {X 0,Y 523.964,Z 356.217,A -85,B 0,C 180,E1 -4662.837,E2 -4662.837} C_VEL
LIN {X 0,Y 523.996,Z 356.216,A -85,B 0,C 180,E1 -4665.236,E2 -4665.236} C_VEL
LIN {X 0,Y 524.003,Z 356.21,A -85,B 0,C 180,E1 -4668.394,E2 -4668.394} C_VEL
LIN {X 0,Y 524,Z 356.214,A -85,B 0,C 180,E1 -4671.516,E2 -4671.516} C_VEL
LIN {X 0,Y 524.078,Z 356.203,A -85,B 0,C 180,E1 -4674.613,E2 -4674.613} C_VEL
LIN {X 0,Y 524.104,Z 356.198,A -85,B 0,C 180,E1 -4677.694,E2 -4677.694} C_VEL
LIN {X 0,Y 524.119,Z 356.201,A -85,B 0,C 180,E1 -4680.768,E2 -4680.768} C_VEL
LIN {X 0,Y 524.069,Z 356.207,A -85,B 0,C 180,E1 -4683.075,E2 -4683.075} C_VEL
LIN {X 0,Y 524.038,Z 356.206,A -85,B 0,C 180,E1 -4686.159,E2 -4686.159} C_VEL
LIN {X 0,Y 523.996,Z 356.214,A -85,B 0,C 180,E1 -4689.262,E2 -4689.262} C_VEL
LIN {X 0,Y 524.015,Z 356.208,A -85,B 0,C 180,E1 -4691.751,E2 -4691.751} C_VEL
LIN {X 0,Y 523.984,Z 356.216,A -85,B 0,C 180,E1 -4695.053,E2 -4695.053} C_VEL
LIN {X 0,Y 523.955,Z 356.216,A -85,B 0,C 180,E1 -4697.969,E2 -4697.969} C_VEL
LIN {X 0,Y 523.965,Z 356.22,A -85,B 0,C 180,E1 -4700.41,E2 -4700.41} C_VEL
LIN {X 0,Y 523.936,Z 356.222,A -85,B 0,C 180,E1 -4702.892,E2 -4702.892} C_VEL
LIN {X 0,Y 523.978,Z 356.215,A -85,B 0,C 180,E1 -4706.021,E2 -4706.021} C_VEL
LIN {X 0,Y 523.933,Z 356.222,A -85,B 0,C 180,E1 -4708.875,E2 -4708.875} C_VEL
LIN {X 0,Y 523.924,Z 356.219,A -85,B 0,C 180,E1 -4711.544,E2 -4711.544} C_VEL
LIN {X 0,Y 523.939,Z 356.225,A -85,B 0,C 180,E1 -4714.29,E2 -4714.29} C_VEL
LIN {X 0,Y 523.907,Z 356.221,A -85,B 0,C 180,E1 -4717.132,E2 -4717.132} C_VEL
LIN {X 0,Y 523.963,Z 356.221,A -85,B 0,C 180,E1 -4720.135,E2 -4720.135} C_VEL
LIN {X 0,Y 523.92,Z 356.219,A -85,B 0,C 180,E1 -4723.167,E2 -4723.167} C_VEL
LIN {X 0,Y 523.937,Z 356.22,A -85,B 0,C 180,E1 -4725.773,E2 -4725.773} C_VEL
LIN {X 0,Y 523.941,Z 356.217,A -85,B 0,C 180,E1 -4728.909,E2 -4728.909} C_VEL
LIN {X 0,Y 523.915,Z 356.226,A -85,B 0,C 180,E1 -4731.899,E2 -4731.899} C_VEL
LIN {X 0,Y 523.937,Z 356.217,A -85,B 0,C 180,E1 -4734.909,E2 -4734.909} C_VEL
LIN {X 0,Y 523.942,Z 356.221,A -85,B 0,C 180,E1 -4737.679,E2 -4737.679} C_VEL
LIN {X 0,Y 523.97,Z 356.214,A -85,B 0,C 180,E1 -4740.674,E2 -4740.674} C_VEL
LIN {X 0,Y 523.975,Z 356.22,A -85,B 0,C 180,E1 -4743.729,E2 -4743.729} C_VEL
LIN {X 0,Y 524.031,Z 356.349,A -85,B 0,C 180,E1 -4744.931,E2 -4744.931} C_VEL
LIN {X 0,Y 525.592,Z 365.006,A -85,B 0,C 180,E1 -4746.351,E2 -4746.351} C_VEL
LIN {X 0,Y 525.178,Z 382.523,A -85,B 0,C 180,E1 -4749.025,E2 -4749.025} C_VEL
LIN {X 0,Y 524.683,Z 404.072,A -85,B 0,C 180,E1 -4752.258,E2 -4752.258} C_VEL
LIN {X 0,Y 524.335,Z 421.49,A -85,B 0,C 180,E1 -4754.839,E2 -4754.839} C_VEL
LIN {X 0,Y 525.962,Z 432.969,A -85,B 0,C 180,E1 -4755.047,E2 -4755.047} C_VEL
LIN {X 0,Y 525.539,Z 530.018,A -85,B 0,C 180,E1 -4756.392,E2 -4756.392} C_VEL
LIN {X 0,Y 525.275,Z 543.325,A -85,B 0,C 180,E1 -4756.73,E2 -4756.73} C_VEL
LIN {X 0,Y 525.018,Z 556.645,A -85,B 0,C 180,E1 -4757.24,E2 -4757.24} C_VEL
LIN {X 0,Y 524.714,Z 568.992,A -85,B 0,C 180,E1 -4757.894,E2 -4757.894} C_VEL
LIN {X 0,Y 524.474,Z 580.757,A -85,B 0,C 180,E1 -4758.699,E2 -4758.699} C_VEL
LIN {X 0,Y 524.166,Z 590.981,A -85,B 0,C 180,E1 -4759.572,E2 -4759.572} C_VEL
LIN {X 0,Y 523.953,Z 600.186,A -85,B 0,C 180,E1 -4760.543,E2 -4760.543} C_VEL
LIN {X 0,Y 523.732,Z 609.156,A -85,B 0,C 180,E1 -4761.706,E2 -4761.706} C_VEL
LIN {X 0,Y 523.583,Z 616.379,A -85,B 0,C 180,E1 -4762.868,E2 -4762.868} C_VEL
LIN {X 0,Y 523.508,Z 622.96,A -85,B 0,C 180,E1 -4764.221,E2 -4764.221} C_VEL
LIN {X 0,Y 523.36,Z 627.309,A -85,B 0,C 180,E1 -4765.379,E2 -4765.379} C_VEL
LIN {X 0,Y 523.443,Z 629.618,A -85,B 0,C 180,E1 -4766.151,E2 -4766.151} C_VEL
LIN {X 0,Y 523.367,Z 631.484,A -85,B 0,C 180,E1 -4766.921,E2 -4766.921} C_VEL
LIN {X 0,Y 523.334,Z 632.884,A -85,B 0,C 180,E1 -4767.691,E2 -4767.691} C_VEL
LIN {X 0,Y 523.25,Z 634.49,A -85,B 0,C 180,E1 -4769.23,E2 -4769.23} C_VEL
LIN {X 0,Y 523.249,Z 634.707,A -85,B 0,C 180,E1 -4770,E2 -4770} C_VEL
LIN {X 0,Y 523.274,Z 633.881,A -85,B 0,C 180,E1 -4771.539,E2 -4771.539} C_VEL
LIN {X 0,Y 523.334,Z 632.885,A -85,B 0,C 180,E1 -4772.309,E2 -4772.309} C_VEL
LIN {X 0,Y 523.367,Z 631.485,A -85,B 0,C 180,E1 -4773.079,E2 -4773.079} C_VEL
LIN {X 0,Y 523.424,Z 628.539,A -85,B 0,C 180,E1 -4774.235,E2 -4774.235} C_VEL
LIN {X 0,Y 523.461,Z 624.55,A -85,B 0,C 180,E1 -4775.393,E2 -4775.393} C_VEL
LIN {X 0,Y 523.517,Z 619.302,A -85,B 0,C 180,E1 -4776.576,E2 -4776.576} C_VEL
LIN {X 0,Y 523.651,Z 612.957,A -85,B 0,C 180,E1 -4777.713,E2 -4777.713} C_VEL
LIN {X 0,Y 523.835,Z 604.9,A -85,B 0,C 180,E1 -4778.875,E2 -4778.875} C_VEL
LIN {X 0,Y 524.034,Z 596.692,A -85,B 0,C 180,E1 -4779.845,E2 -4779.845} C_VEL
LIN {X 0,Y 524.344,Z 586.689,A -85,B 0,C 180,E1 -4780.815,E2 -4780.815} C_VEL
LIN {X 0,Y 524.561,Z 575.426,A -85,B 0,C 180,E1 -4781.689,E2 -4781.689} C_VEL
LIN {X 0,Y 524.861,Z 564.336,A -85,B 0,C 180,E1 -4782.371,E2 -4782.371} C_VEL
LIN {X 0,Y 525.107,Z 552.084,A -85,B 0,C 180,E1 -4782.954,E2 -4782.954} C_VEL
LIN {X 0,Y 525.349,Z 539.235,A -85,B 0,C 180,E1 -4783.391,E2 -4783.391} C_VEL
LIN {X 0,Y 525.563,Z 525.619,A -85,B 0,C 180,E1 -4783.681,E2 -4783.681} C_VEL
LIN {X 0,Y 525.809,Z 431.141,A -85,B 0,C 180,E1 -4784.982,E2 -4784.982} C_VEL
LIN {X 0,Y 524.314,Z 421.416,A -85,B 0,C 180,E1 -4785.167,E2 -4785.167} C_VEL
LIN {X 0,Y 524.734,Z 400.241,A -85,B 0,C 180,E1 -4788.305,E2 -4788.305} C_VEL
LIN {X 0,Y 525.175,Z 381.096,A -85,B 0,C 180,E1 -4791.181,E2 -4791.181} C_VEL
LIN {X 0,Y 525.61,Z 364.926,A -85,B 0,C 180,E1 -4793.648,E2 -4793.648} C_VEL
LIN {X 0,Y 524.029,Z 356.21,A -85,B 0,C 180,E1 -4795.095,E2 -4795.095} C_VEL
LIN {X 0,Y 523.97,Z 356.22,A -85,B 0,C 180,E1 -4797.998,E2 -4797.998} C_VEL
LIN {X 0,Y 523.952,Z 356.214,A -85,B 0,C 180,E1 -4800.856,E2 -4800.856} C_VEL
LIN {X 0,Y 523.96,Z 356.22,A -85,B 0,C 180,E1 -4803.734,E2 -4803.734} C_VEL
LIN {X 0,Y 523.921,Z 356.222,A -85,B 0,C 180,E1 -4806.404,E2 -4806.404} C_VEL
LIN {X 0,Y 523.921,Z 356.219,A -85,B 0,C 180,E1 -4809.084,E2 -4809.084} C_VEL
LIN {X 0,Y 523.953,Z 356.218,A -85,B 0,C 180,E1 -4812.118,E2 -4812.118} C_VEL
LIN {X 0,Y 523.951,Z 356.216,A -85,B 0,C 180,E1 -4815.308,E2 -4815.308} C_VEL
LIN {X 0,Y 523.967,Z 356.211,A -85,B 0,C 180,E1 -4818.687,E2 -4818.687} C_VEL
LIN {X 0,Y 523.92,Z 356.219,A -85,B 0,C 180,E1 -4821.079,E2 -4821.079} C_VEL
LIN {X 0,Y 523.924,Z 356.223,A -85,B 0,C 180,E1 -4823.827,E2 -4823.827} C_VEL
LIN {X 0,Y 523.937,Z 356.216,A -85,B 0,C 180,E1 -4826.635,E2 -4826.635} C_VEL
LIN {X 0,Y 523.956,Z 356.221,A -85,B 0,C 180,E1 -4829.356,E2 -4829.356} C_VEL
LIN {X 0,Y 523.972,Z 356.212,A -85,B 0,C 180,E1 -4832.28,E2 -4832.28} C_VEL
LIN {X 0,Y 523.948,Z 356.21,A -85,B 0,C 180,E1 -4834.581,E2 -4834.581} C_VEL
LIN {X 0,Y 523.936,Z 356.219,A -85,B 0,C 180,E1 -4837.108,E2 -4837.108} C_VEL
LIN {X 0,Y 523.97,Z 356.212,A -85,B 0,C 180,E1 -4839.865,E2 -4839.865} C_VEL
LIN {X 0,Y 523.963,Z 356.217,A -85,B 0,C 180,E1 -4842.837,E2 -4842.837} C_VEL
LIN {X 0,Y 523.967,Z 356.219,A -85,B 0,C 180,E1 -4845.236,E2 -4845.236} C_VEL
LIN {X 0,Y 524.003,Z 356.209,A -85,B 0,C 180,E1 -4848.394,E2 -4848.394} C_VEL
LIN {X 0,Y 524,Z 356.211,A -85,B 0,C 180,E1 -4851.516,E2 -4851.516} C_VEL
LIN {X 0,Y 524.077,Z 356.2,A -85,B 0,C 180,E1 -4854.614,E2 -4854.614} C_VEL
LIN {X 0,Y 524.104,Z 356.195,A -85,B 0,C 180,E1 -4857.695,E2 -4857.695} C_VEL
LIN {X 0,Y 524.119,Z 356.201,A -85,B 0,C 180,E1 -4860.769,E2 -4860.769} C_VEL
LIN {X 0,Y 524.069,Z 356.203,A -85,B 0,C 180,E1 -4863.075,E2 -4863.075} C_VEL
LIN {X 0,Y 524.038,Z 356.206,A -85,B 0,C 180,E1 -4866.159,E2 -4866.159} C_VEL
